LIN {X 0,Y 228.95,Z 464.335,A -85,B 0,C 180,E1 -20820.068,E2 -20820.068} C_VEL
LIN {X 0,Y 225.783,Z 455.816,A -85,B 0,C 180,E1 -20821.561,E2 -20821.561} C_VEL
LIN {X 0,Y 220.745,Z 444.883,A -85,B 0,C 180,E1 -20823.412,E2 -20823.412} C_VEL
LIN {X 0,Y 215.443,Z 435.104,A -85,B 0,C 180,E1 -20825.049,E2 -20825.049} C_VEL
LIN {X 0,Y 214.125,Z 432.902,A -85,B 0,C 180,E1 -20825.41,E2 -20825.41} C_VEL
LIN {X 0,Y 213.741,Z 431.362,A -85,B 0,C 180,E1 -20825.591,E2 -20825.591} C_VEL
LIN {X 0,Y 213.731,Z 431.362,A -85,B 0,C 180,E1 -20828.664,E2 -20828.664} C_VEL
LIN {X 0,Y 213.704,Z 431.366,A -85,B 0,C 180,E1 -20833.678,E2 -20833.678} C_VEL
LIN {X 0,Y 213.702,Z 431.365,A -85,B 0,C 180,E1 -20836.344,E2 -20836.344} C_VEL
LIN {X 0,Y 213.712,Z 431.364,A -85,B 0,C 180,E1 -20839.143,E2 -20839.143} C_VEL
LIN {X 0,Y 213.738,Z 431.359,A -85,B 0,C 180,E1 -20843.712,E2 -20843.712} C_VEL
LIN {X 0,Y 213.79,Z 431.354,A -85,B 0,C 180,E1 -20848.725,E2 -20848.725} C_VEL
LIN {X 0,Y 213.821,Z 431.351,A -85,B 0,C 180,E1 -20852.604,E2 -20852.604} C_VEL
LIN {X 0,Y 213.847,Z 431.347,A -85,B 0,C 180,E1 -20856.954,E2 -20856.954} C_VEL
LIN {X 0,Y 213.957,Z 431.335,A -85,B 0,C 180,E1 -20862.806,E2 -20862.806} C_VEL
LIN {X 0,Y 213.947,Z 431.333,A -85,B 0,C 180,E1 -20866.707,E2 -20866.707} C_VEL
LIN {X 0,Y 214.137,Z 431.305,A -85,B 0,C 180,E1 -20870.556,E2 -20870.556} C_VEL
LIN {X 0,Y 214.096,Z 431.314,A -85,B 0,C 180,E1 -20874.349,E2 -20874.349} C_VEL
LIN {X 0,Y 214.44,Z 431.245,A -85,B 0,C 180,E1 -20878.123,E2 -20878.123} C_VEL
LIN {X 0,Y 214.545,Z 431.244,A -85,B 0,C 180,E1 -20880.001,E2 -20880.001} C_VEL
LIN {X 0,Y 214.441,Z 431.269,A -85,B 0,C 180,E1 -20881.879,E2 -20881.879} C_VEL
LIN {X 0,Y 214.194,Z 431.304,A -85,B 0,C 180,E1 -20887.543,E2 -20887.543} C_VEL
LIN {X 0,Y 213.995,Z 431.329,A -85,B 0,C 180,E1 -20891.366,E2 -20891.366} C_VEL
LIN {X 0,Y 213.926,Z 431.338,A -85,B 0,C 180,E1 -20895.238,E2 -20895.238} C_VEL
LIN {X 0,Y 213.832,Z 431.349,A -85,B 0,C 180,E1 -20899.189,E2 -20899.189} C_VEL
LIN {X 0,Y 213.809,Z 431.355,A -85,B 0,C 180,E1 -20903.232,E2 -20903.232} C_VEL
LIN {X 0,Y 213.846,Z 431.557,A -85,B 0,C 180,E1 -20907.461,E2 -20907.461} C_VEL
LIN {X 0,Y 214.012,Z 433.205,A -85,B 0,C 180,E1 -20911.698,E2 -20911.698} C_VEL
LIN {X 0,Y 214.268,Z 435.135,A -85,B 0,C 180,E1 -20916.187,E2 -20916.187} C_VEL
LIN {X 0,Y 214.637,Z 437.558,A -85,B 0,C 180,E1 -20921.142,E2 -20921.142} C_VEL
LIN {X 0,Y 214.751,Z 439.049,A -85,B 0,C 180,E1 -20923.949,E2 -20923.949} C_VEL
LIN {X 0,Y 214.709,Z 440.54,A -85,B 0,C 180,E1 -20926.578,E2 -20926.578} C_VEL
LIN {X 0,Y 214.485,Z 442.03,A -85,B 0,C 180,E1 -20929.056,E2 -20929.056} C_VEL
LIN {X 0,Y 214.086,Z 443.875,A -85,B 0,C 180,E1 -20931.988,E2 -20931.988} C_VEL
LIN {X 0,Y 213.633,Z 445.658,A -85,B 0,C 180,E1 -20934.669,E2 -20934.669} C_VEL
LIN {X 0,Y 214.482,Z 448.767,A -85,B 0,C 180,E1 -20935.005,E2 -20935.005} C_VEL
LIN {X 0,Y 216.666,Z 454.962,A -85,B 0,C 180,E1 -20935.878,E2 -20935.878} C_VEL
LIN {X 0,Y 219.161,Z 463.344,A -85,B 0,C 180,E1 -20937.069,E2 -20937.069} C_VEL
LIN {X 0,Y 221.554,Z 473.865,A -85,B 0,C 180,E1 -20938.668,E2 -20938.668} C_VEL
LIN {X 0,Y 222.983,Z 483.529,A -85,B 0,C 180,E1 -20940.26,E2 -20940.26} C_VEL
LIN {X 0,Y 223.821,Z 492.472,A -85,B 0,C 180,E1 -20941.901,E2 -20941.901} C_VEL
LIN {X 0,Y 223.91,Z 501.294,A -85,B 0,C 180,E1 -20943.689,E2 -20943.689} C_VEL
LIN {X 0,Y 223.656,Z 504.689,A -85,B 0,C 180,E1 -20944.402,E2 -20944.402} C_VEL
LIN {X 0,Y 220.986,Z 514.268,A -85,B 0,C 180,E1 -20946.576,E2 -20946.576} C_VEL
LIN {X 0,Y 218.846,Z 521.593,A -85,B 0,C 180,E1 -20948.641,E2 -20948.641} C_VEL
LIN {X 0,Y 216.772,Z 528.635,A -85,B 0,C 180,E1 -20951.083,E2 -20951.083} C_VEL
LIN {X 0,Y 215.461,Z 533.139,A -85,B 0,C 180,E1 -20952.929,E2 -20952.929} C_VEL
LIN {X 0,Y 213.707,Z 538.674,A -85,B 0,C 180,E1 -20955.749,E2 -20955.749} C_VEL
LIN {X 0,Y 212.4,Z 541.079,A -85,B 0,C 180,E1 -20957.173,E2 -20957.173} C_VEL
LIN {X 0,Y 208.716,Z 544.319,A -85,B 0,C 180,E1 -20959.521,E2 -20959.521} C_VEL
LIN {X 0,Y 205.844,Z 546.363,A -85,B 0,C 180,E1 -20961.49,E2 -20961.49} C_VEL
LIN {X 0,Y 204.575,Z 547.716,A -85,B 0,C 180,E1 -20963.064,E2 -20963.064} C_VEL
LIN {X 0,Y 204.437,Z 547.992,A -85,B 0,C 180,E1 -20963.604,E2 -20963.604} C_VEL
LIN {X 0,Y 204.339,Z 549.391,A -85,B 0,C 180,E1 -20966.056,E2 -20966.056} C_VEL
LIN {X 0,Y 204.335,Z 549.984,A -85,B 0,C 180,E1 -20968.029,E2 -20968.029} C_VEL
LIN {X 0,Y 204.444,Z 550.143,A -85,B 0,C 180,E1 -20970,E2 -20970} C_VEL
LIN {X 0,Y 204.334,Z 549.984,A -85,B 0,C 180,E1 -20971.971,E2 -20971.971} C_VEL
LIN {X 0,Y 204.299,Z 549.39,A -85,B 0,C 180,E1 -20973.945,E2 -20973.945} C_VEL
LIN {X 0,Y 204.645,Z 546.935,A -85,B 0,C 180,E1 -20977.895,E2 -20977.895} C_VEL
LIN {X 0,Y 205.321,Z 543.98,A -85,B 0,C 180,E1 -20980.851,E2 -20980.851} C_VEL
LIN {X 0,Y 206.335,Z 539.986,A -85,B 0,C 180,E1 -20983.793,E2 -20983.793} C_VEL
LIN {X 0,Y 207.988,Z 534.856,A -85,B 0,C 180,E1 -20986.691,E2 -20986.691} C_VEL
LIN {X 0,Y 209.661,Z 529.593,A -85,B 0,C 180,E1 -20989.076,E2 -20989.076} C_VEL
LIN {X 0,Y 211.328,Z 524.655,A -85,B 0,C 180,E1 -20990.947,E2 -20990.947} C_VEL
LIN {X 0,Y 213.4,Z 517.322,A -85,B 0,C 180,E1 -20993.278,E2 -20993.278} C_VEL
LIN {X 0,Y 215.512,Z 510.399,A -85,B 0,C 180,E1 -20995.083,E2 -20995.083} C_VEL
LIN {X 0,Y 217.206,Z 504.49,A -85,B 0,C 180,E1 -20996.416,E2 -20996.416} C_VEL
LIN {X 0,Y 217.303,Z 494.811,A -85,B 0,C 180,E1 -20998.526,E2 -20998.526} C_VEL
LIN {X 0,Y 216.575,Z 485.637,A -85,B 0,C 180,E1 -21000.333,E2 -21000.333} C_VEL
LIN {X 0,Y 215.38,Z 476.429,A -85,B 0,C 180,E1 -21001.96,E2 -21001.96} C_VEL
LIN {X 0,Y 213.251,Z 466.398,A -85,B 0,C 180,E1 -21003.609,E2 -21003.609} C_VEL
LIN {X 0,Y 210.509,Z 456.533,A -85,B 0,C 180,E1 -21005.117,E2 -21005.117} C_VEL
LIN {X 0,Y 207.828,Z 448.996,A -85,B 0,C 180,E1 -21006.261,E2 -21006.261} C_VEL
LIN {X 0,Y 206.874,Z 446.301,A -85,B 0,C 180,E1 -21006.61,E2 -21006.61} C_VEL
LIN {X 0,Y 206.779,Z 445.482,A -85,B 0,C 180,E1 -21006.726,E2 -21006.726} C_VEL
LIN {X 0,Y 207.262,Z 443.315,A -85,B 0,C 180,E1 -21010.11,E2 -21010.11} C_VEL
LIN {X 0,Y 207.548,Z 441.811,A -85,B 0,C 180,E1 -21012.627,E2 -21012.627} C_VEL
LIN {X 0,Y 207.693,Z 440.333,A -85,B 0,C 180,E1 -21015.283,E2 -21015.283} C_VEL
LIN {X 0,Y 207.5,Z 437.944,A -85,B 0,C 180,E1 -21019.943,E2 -21019.943} C_VEL
LIN {X 0,Y 207.199,Z 435.719,A -85,B 0,C 180,E1 -21024.785,E2 -21024.785} C_VEL
LIN {X 0,Y 206.948,Z 433.839,A -85,B 0,C 180,E1 -21029.375,E2 -21029.375} C_VEL
LIN {X 0,Y 206.73,Z 432.247,A -85,B 0,C 180,E1 -21033.771,E2 -21033.771} C_VEL
LIN {X 0,Y 206.736,Z 432.236,A -85,B 0,C 180,E1 -21038.04,E2 -21038.04} C_VEL
LIN {X 0,Y 206.87,Z 432.218,A -85,B 0,C 180,E1 -21042.195,E2 -21042.195} C_VEL
LIN {X 0,Y 206.889,Z 432.214,A -85,B 0,C 180,E1 -21046.243,E2 -21046.243} C_VEL
LIN {X 0,Y 207.096,Z 432.188,A -85,B 0,C 180,E1 -21050.23,E2 -21050.23} C_VEL
LIN {X 0,Y 207.058,Z 432.192,A -85,B 0,C 180,E1 -21054.155,E2 -21054.155} C_VEL
LIN {X 0,Y 207.378,Z 432.149,A -85,B 0,C 180,E1 -21058.057,E2 -21058.057} C_VEL
LIN {X 0,Y 207.51,Z 432.119,A -85,B 0,C 180,E1 -21059.999,E2 -21059.999} C_VEL
LIN {X 0,Y 207.377,Z 432.124,A -85,B 0,C 180,E1 -21061.941,E2 -21061.941} C_VEL
LIN {X 0,Y 207.144,Z 432.18,A -85,B 0,C 180,E1 -21067.799,E2 -21067.799} C_VEL
LIN {X 0,Y 206.919,Z 432.21,A -85,B 0,C 180,E1 -21071.758,E2 -21071.758} C_VEL
LIN {X 0,Y 206.866,Z 432.214,A -85,B 0,C 180,E1 -21075.77,E2 -21075.77} C_VEL
LIN {X 0,Y 206.779,Z 432.22,A -85,B 0,C 180,E1 -21079.868,E2 -21079.868} C_VEL
LIN {X 0,Y 206.759,Z 432.226,A -85,B 0,C 180,E1 -21084.071,E2 -21084.071} C_VEL
LIN {X 0,Y 206.739,Z 432.232,A -85,B 0,C 180,E1 -21088.418,E2 -21088.418} C_VEL
LIN {X 0,Y 206.704,Z 432.237,A -85,B 0,C 180,E1 -21092.955,E2 -21092.955} C_VEL
LIN {X 0,Y 206.721,Z 432.233,A -85,B 0,C 180,E1 -21097.73,E2 -21097.73} C_VEL
LIN {X 0,Y 206.721,Z 432.235,A -85,B 0,C 180,E1 -21101.589,E2 -21101.589} C_VEL
LIN {X 0,Y 206.669,Z 432.241,A -85,B 0,C 180,E1 -21105.57,E2 -21105.57} C_VEL
LIN {X 0,Y 206.669,Z 432.24,A -85,B 0,C 180,E1 -21109.752,E2 -21109.752} C_VEL
LIN {X 0,Y 206.71,Z 432.237,A -85,B 0,C 180,E1 -21113.049,E2 -21113.049} C_VEL
LIN {X 0,Y 207.757,Z 435.179,A -85,B 0,C 180,E1 -21113.464,E2 -21113.464} C_VEL
LIN {X 0,Y 209.142,Z 437.168,A -85,B 0,C 180,E1 -21113.858,E2 -21113.858} C_VEL
LIN {X 0,Y 214.876,Z 447.881,A -85,B 0,C 180,E1 -21115.778,E2 -21115.778} C_VEL
LIN {X 0,Y 220.603,Z 460.836,A -85,B 0,C 180,E1 -21118.167,E2 -21118.167} C_VEL
LIN {X 0,Y 223.937,Z 470.772,A -85,B 0,C 180,E1 -21120.071,E2 -21120.071} C_VEL
LIN {X 0,Y 226.919,Z 479.248,A -85,B 0,C 180,E1 -21121.902,E2 -21121.902} C_VEL
LIN {X 0,Y 230.977,Z 487.85,A -85,B 0,C 180,E1 -21124.091,E2 -21124.091} C_VEL
LIN {X 0,Y 235.85,Z 495.643,A -85,B 0,C 180,E1 -21126.388,E2 -21126.388} C_VEL
LIN {X 0,Y 242.584,Z 503.921,A -85,B 0,C 180,E1 -21129.183,E2 -21129.183} C_VEL
LIN {X 0,Y 250.878,Z 511.914,A -85,B 0,C 180,E1 -21132.259,E2 -21132.259} C_VEL
LIN {X 0,Y 258.464,Z 517.884,A -85,B 0,C 180,E1 -21134.854,E2 -21134.854} C_VEL
LIN {X 0,Y 267.452,Z 523.982,A -85,B 0,C 180,E1 -21137.865,E2 -21137.865} C_VEL
LIN {X 0,Y 274.679,Z 528.41,A -85,B 0,C 180,E1 -21140.427,E2 -21140.427} C_VEL
LIN {X 0,Y 280.649,Z 531.794,A -85,B 0,C 180,E1 -21142.807,E2 -21142.807} C_VEL
LIN {X 0,Y 283.647,Z 533.508,A -85,B 0,C 180,E1 -21144.312,E2 -21144.312} C_VEL
LIN {X 0,Y 285.796,Z 534.827,A -85,B 0,C 180,E1 -21145.769,E2 -21145.769} C_VEL
LIN {X 0,Y 288.397,Z 535.966,A -85,B 0,C 180,E1 -21147.597,E2 -21147.597} C_VEL
LIN {X 0,Y 289.489,Z 536.314,A -85,B 0,C 180,E1 -21148.609,E2 -21148.609} C_VEL
LIN {X 0,Y 290.513,Z 536.484,A -85,B 0,C 180,E1 -21150,E2 -21150} C_VEL
LIN {X 0,Y 289.482,Z 536.314,A -85,B 0,C 180,E1 -21151.391,E2 -21151.391} C_VEL
LIN {X 0,Y 287.845,Z 535.767,A -85,B 0,C 180,E1 -21152.799,E2 -21152.799} C_VEL
LIN {X 0,Y 285.796,Z 534.827,A -85,B 0,C 180,E1 -21154.231,E2 -21154.231} C_VEL
LIN {X 0,Y 282.767,Z 532.973,A -85,B 0,C 180,E1 -21156.196,E2 -21156.196} C_VEL
LIN {X 0,Y 280.611,Z 531.795,A -85,B 0,C 180,E1 -21157.194,E2 -21157.194} C_VEL
LIN {X 0,Y 274.692,Z 528.41,A -85,B 0,C 180,E1 -21159.573,E2 -21159.573} C_VEL
LIN {X 0,Y 267.467,Z 523.982,A -85,B 0,C 180,E1 -21162.134,E2 -21162.134} C_VEL
LIN {X 0,Y 258.459,Z 517.897,A -85,B 0,C 180,E1 -21165.142,E2 -21165.142} C_VEL
LIN {X 0,Y 250.189,Z 511.27,A -85,B 0,C 180,E1 -21167.998,E2 -21167.998} C_VEL
LIN {X 0,Y 242.6,Z 503.901,A -85,B 0,C 180,E1 -21170.821,E2 -21170.821} C_VEL
LIN {X 0,Y 235.851,Z 495.641,A -85,B 0,C 180,E1 -21173.612,E2 -21173.612} C_VEL
LIN {X 0,Y 230.442,Z 486.799,A -85,B 0,C 180,E1 -21176.187,E2 -21176.187} C_VEL
LIN {X 0,Y 226.499,Z 478.07,A -85,B 0,C 180,E1 -21178.368,E2 -21178.368} C_VEL
LIN {X 0,Y 222.715,Z 466.813,A -85,B 0,C 180,E1 -21180.697,E2 -21180.697} C_VEL
LIN {X 0,Y 219.268,Z 457.558,A -85,B 0,C 180,E1 -21182.446,E2 -21182.446} C_VEL
LIN {X 0,Y 214.039,Z 446.14,A -85,B 0,C 180,E1 -21184.519,E2 -21184.519} C_VEL
LIN {X 0,Y 208.408,Z 436.025,A -85,B 0,C 180,E1 -21186.376,E2 -21186.376} C_VEL
LIN {X 0,Y 206.986,Z 433.495,A -85,B 0,C 180,E1 -21186.81,E2 -21186.81} C_VEL
LIN {X 0,Y 206.695,Z 432.239,A -85,B 0,C 180,E1 -21186.946,E2 -21186.946} C_VEL
LIN {X 0,Y 206.641,Z 432.246,A -85,B 0,C 180,E1 -21191.564,E2 -21191.564} C_VEL
LIN {X 0,Y 206.63,Z 432.247,A -85,B 0,C 180,E1 -21195.582,E2 -21195.582} C_VEL
LIN {X 0,Y 206.655,Z 432.243,A -85,B 0,C 180,E1 -21199.749,E2 -21199.749} C_VEL
LIN {X 0,Y 206.694,Z 432.237,A -85,B 0,C 180,E1 -21204.689,E2 -21204.689} C_VEL
LIN {X 0,Y 206.718,Z 432.236,A -85,B 0,C 180,E1 -21209.34,E2 -21209.34} C_VEL
LIN {X 0,Y 206.728,Z 432.231,A -85,B 0,C 180,E1 -21213.773,E2 -21213.773} C_VEL
LIN {X 0,Y 206.753,Z 432.23,A -85,B 0,C 180,E1 -21218.044,E2 -21218.044} C_VEL
LIN {X 0,Y 206.868,Z 432.215,A -85,B 0,C 180,E1 -21222.197,E2 -21222.197} C_VEL
LIN {X 0,Y 206.889,Z 432.209,A -85,B 0,C 180,E1 -21226.245,E2 -21226.245} C_VEL
LIN {X 0,Y 207.095,Z 432.182,A -85,B 0,C 180,E1 -21230.232,E2 -21230.232} C_VEL
LIN {X 0,Y 207.057,Z 432.193,A -85,B 0,C 180,E1 -21234.157,E2 -21234.157} C_VEL
LIN {X 0,Y 207.377,Z 432.124,A -85,B 0,C 180,E1 -21238.059,E2 -21238.059} C_VEL
LIN {X 0,Y 207.51,Z 432.119,A -85,B 0,C 180,E1 -21240.001,E2 -21240.001} C_VEL
LIN {X 0,Y 207.378,Z 432.149,A -85,B 0,C 180,E1 -21241.943,E2 -21241.943} C_VEL
LIN {X 0,Y 207.137,Z 432.183,A -85,B 0,C 180,E1 -21247.801,E2 -21247.801} C_VEL
LIN {X 0,Y 206.92,Z 432.211,A -85,B 0,C 180,E1 -21251.76,E2 -21251.76} C_VEL
LIN {X 0,Y 206.861,Z 432.22,A -85,B 0,C 180,E1 -21255.772,E2 -21255.772} C_VEL
LIN {X 0,Y 206.775,Z 432.229,A -85,B 0,C 180,E1 -21259.871,E2 -21259.871} C_VEL
LIN {X 0,Y 206.745,Z 432.238,A -85,B 0,C 180,E1 -21264.076,E2 -21264.076} C_VEL
LIN {X 0,Y 206.73,Z 432.253,A -85,B 0,C 180,E1 -21266.229,E2 -21266.229} C_VEL
LIN {X 0,Y 206.948,Z 433.841,A -85,B 0,C 180,E1 -21270.625,E2 -21270.625} C_VEL
LIN {X 0,Y 207.206,Z 435.844,A -85,B 0,C 180,E1 -21275.51,E2 -21275.51} C_VEL
LIN {X 0,Y 207.505,Z 437.945,A -85,B 0,C 180,E1 -21280.055,E2 -21280.055} C_VEL
LIN {X 0,Y 207.632,Z 439.227,A -85,B 0,C 180,E1 -21282.608,E2 -21282.608} C_VEL
LIN {X 0,Y 207.678,Z 440.668,A -85,B 0,C 180,E1 -21285.29,E2 -21285.29} C_VEL
LIN {X 0,Y 207.479,Z 442.319,A -85,B 0,C 180,E1 -21288.179,E2 -21288.179} C_VEL
LIN {X 0,Y 206.932,Z 444.794,A -85,B 0,C 180,E1 -21292.315,E2 -21292.315} C_VEL
LIN {X 0,Y 206.779,Z 445.439,A -85,B 0,C 180,E1 -21293.275,E2 -21293.275} C_VEL
LIN {X 0,Y 207.828,Z 448.982,A -85,B 0,C 180,E1 -21293.738,E2 -21293.738} C_VEL
LIN {X 0,Y 211.592,Z 459.902,A -85,B 0,C 180,E1 -21295.378,E2 -21295.378} C_VEL
LIN {X 0,Y 214.365,Z 471.313,A -85,B 0,C 180,E1 -21297.172,E2 -21297.172} C_VEL
LIN {X 0,Y 216.106,Z 481.185,A -85,B 0,C 180,E1 -21298.862,E2 -21298.862} C_VEL
LIN {X 0,Y 217.044,Z 490.271,A -85,B 0,C 180,E1 -21300.554,E2 -21300.554} C_VEL
LIN {X 0,Y 217.32,Z 498.233,A -85,B 0,C 180,E1 -21302.174,E2 -21302.174} C_VEL
LIN {X 0,Y 216.968,Z 505.58,A -85,B 0,C 180,E1 -21303.811,E2 -21303.811} C_VEL
LIN {X 0,Y 214.482,Z 514.07,A -85,B 0,C 180,E1 -21305.821,E2 -21305.821} C_VEL
LIN {X 0,Y 212.042,Z 521.97,A -85,B 0,C 180,E1 -21308.134,E2 -21308.134} C_VEL
LIN {X 0,Y 210.053,Z 528.438,A -85,B 0,C 180,E1 -21310.453,E2 -21310.453} C_VEL
LIN {X 0,Y 208.659,Z 532.941,A -85,B 0,C 180,E1 -21312.354,E2 -21312.354} C_VEL
LIN {X 0,Y 206.707,Z 538.795,A -85,B 0,C 180,E1 -21315.462,E2 -21315.462} C_VEL
LIN {X 0,Y 205.611,Z 542.761,A -85,B 0,C 180,E1 -21318.166,E2 -21318.166} C_VEL
LIN {X 0,Y 205.071,Z 545.133,A -85,B 0,C 180,E1 -21320.134,E2 -21320.134} C_VEL
LIN {X 0,Y 204.437,Z 547.992,A -85,B 0,C 180,E1 -21323.604,E2 -21323.604} C_VEL
LIN {X 0,Y 203.673,Z 549.008,A -85,B 0,C 180,E1 -21325.226,E2 -21325.226} C_VEL
LIN {X 0,Y 202.069,Z 549.675,A -85,B 0,C 180,E1 -21326.833,E2 -21326.833} C_VEL
LIN {X 0,Y 198.386,Z 550.084,A -85,B 0,C 180,E1 -21330.102,E2 -21330.102} C_VEL
LIN {X 0,Y 197.324,Z 549.856,A -85,B 0,C 180,E1 -21331.809,E2 -21331.809} C_VEL
LIN {X 0,Y 197.219,Z 549.687,A -85,B 0,C 180,E1 -21332.386,E2 -21332.386} C_VEL
LIN {X 0,Y 197.21,Z 549.193,A -85,B 0,C 180,E1 -21334.087,E2 -21334.087} C_VEL
LIN {X 0,Y 197.595,Z 546.737,A -85,B 0,C 180,E1 -21338.179,E2 -21338.179} C_VEL
LIN {X 0,Y 198.307,Z 543.782,A -85,B 0,C 180,E1 -21341.24,E2 -21341.24} C_VEL
LIN {X 0,Y 199.408,Z 539.788,A -85,B 0,C 180,E1 -21344.283,E2 -21344.283} C_VEL
LIN {X 0,Y 201.169,Z 534.658,A -85,B 0,C 180,E1 -21347.274,E2 -21347.274} C_VEL
LIN {X 0,Y 202.94,Z 529.395,A -85,B 0,C 180,E1 -21349.733,E2 -21349.733} C_VEL
LIN {X 0,Y 204.659,Z 524.456,A -85,B 0,C 180,E1 -21351.663,E2 -21351.663} C_VEL
LIN {X 0,Y 206.363,Z 518.752,A -85,B 0,C 180,E1 -21353.587,E2 -21353.587} C_VEL
LIN {X 0,Y 209.076,Z 510.201,A -85,B 0,C 180,E1 -21355.911,E2 -21355.911} C_VEL
LIN {X 0,Y 210.544,Z 505.38,A -85,B 0,C 180,E1 -21357.052,E2 -21357.052} C_VEL
LIN {X 0,Y 210.696,Z 494.601,A -85,B 0,C 180,E1 -21359.508,E2 -21359.508} C_VEL
LIN {X 0,Y 209.952,Z 484.831,A -85,B 0,C 180,E1 -21361.498,E2 -21361.498} C_VEL
LIN {X 0,Y 208.694,Z 476.106,A -85,B 0,C 180,E1 -21363.128,E2 -21363.128} C_VEL
LIN {X 0,Y 206.665,Z 466.416,A -85,B 0,C 180,E1 -21364.804,E2 -21364.804} C_VEL
LIN {X 0,Y 203.784,Z 456.5,A -85,B 0,C 180,E1 -21366.44,E2 -21366.44} C_VEL
LIN {X 0,Y 201.057,Z 448.967,A -85,B 0,C 180,E1 -21367.675,E2 -21367.675} C_VEL
LIN {X 0,Y 200.078,Z 446.209,A -85,B 0,C 180,E1 -21368.061,E2 -21368.061} C_VEL
LIN {X 0,Y 199.968,Z 445.246,A -85,B 0,C 180,E1 -21368.243,E2 -21368.243} C_VEL
LIN {X 0,Y 200.497,Z 442.642,A -85,B 0,C 180,E1 -21372.597,E2 -21372.597} C_VEL
LIN {X 0,Y 200.63,Z 441.069,A -85,B 0,C 180,E1 -21375.524,E2 -21375.524} C_VEL
LIN {X 0,Y 200.566,Z 439.695,A -85,B 0,C 180,E1 -21378.257,E2 -21378.257} C_VEL
LIN {X 0,Y 200.388,Z 438.48,A -85,B 0,C 180,E1 -21380.853,E2 -21380.853} C_VEL
LIN {X 0,Y 200.082,Z 436.327,A -85,B 0,C 180,E1 -21385.804,E2 -21385.804} C_VEL
LIN {X 0,Y 199.872,Z 434.479,A -85,B 0,C 180,E1 -21390.509,E2 -21390.509} C_VEL
LIN {X 0,Y 199.663,Z 433.116,A -85,B 0,C 180,E1 -21395.013,E2 -21395.013} C_VEL
LIN {X 0,Y 199.688,Z 433.113,A -85,B 0,C 180,E1 -21399.392,E2 -21399.392} C_VEL
LIN {X 0,Y 199.799,Z 433.099,A -85,B 0,C 180,E1 -21403.655,E2 -21403.655} C_VEL
LIN {X 0,Y 199.87,Z 433.09,A -85,B 0,C 180,E1 -21407.819,E2 -21407.819} C_VEL
LIN {X 0,Y 200.085,Z 433.061,A -85,B 0,C 180,E1 -21411.922,E2 -21411.922} C_VEL
LIN {X 0,Y 200.317,Z 433.028,A -85,B 0,C 180,E1 -21417.988,E2 -21417.988} C_VEL
LIN {X 0,Y 200.475,Z 432.994,A -85,B 0,C 180,E1 -21419.999,E2 -21419.999} C_VEL
LIN {X 0,Y 200.023,Z 433.053,A -85,B 0,C 180,E1 -21424.028,E2 -21424.028} C_VEL
LIN {X 0,Y 200.091,Z 433.058,A -85,B 0,C 180,E1 -21428.075,E2 -21428.075} C_VEL
LIN {X 0,Y 199.869,Z 433.088,A -85,B 0,C 180,E1 -21432.178,E2 -21432.178} C_VEL
LIN {X 0,Y 199.802,Z 433.095,A -85,B 0,C 180,E1 -21436.342,E2 -21436.342} C_VEL
LIN {X 0,Y 199.695,Z 433.104,A -85,B 0,C 180,E1 -21440.605,E2 -21440.605} C_VEL
LIN {X 0,Y 199.668,Z 433.107,A -85,B 0,C 180,E1 -21444.984,E2 -21444.984} C_VEL
LIN {X 0,Y 199.67,Z 433.114,A -85,B 0,C 180,E1 -21449.522,E2 -21449.522} C_VEL
LIN {X 0,Y 199.659,Z 433.115,A -85,B 0,C 180,E1 -21452.352,E2 -21452.352} C_VEL
LIN {X 0,Y 199.649,Z 433.117,A -85,B 0,C 180,E1 -21456.756,E2 -21456.756} C_VEL
LIN {X 0,Y 199.695,Z 433.111,A -85,B 0,C 180,E1 -21459.306,E2 -21459.306} C_VEL
LIN {X 0,Y 199.659,Z 433.115,A -85,B 0,C 180,E1 -21462.338,E2 -21462.338} C_VEL
LIN {X 0,Y 199.626,Z 433.118,A -85,B 0,C 180,E1 -21465.243,E2 -21465.243} C_VEL
LIN {X 0,Y 199.637,Z 433.118,A -85,B 0,C 180,E1 -21470.756,E2 -21470.756} C_VEL
LIN {X 0,Y 199.672,Z 433.114,A -85,B 0,C 180,E1 -21471.549,E2 -21471.549} C_VEL
LIN {X 0,Y 200.765,Z 436.111,A -85,B 0,C 180,E1 -21472.012,E2 -21472.012} C_VEL
LIN {X 0,Y 202.338,Z 438.455,A -85,B 0,C 180,E1 -21472.497,E2 -21472.497} C_VEL
LIN {X 0,Y 208.631,Z 449.967,A -85,B 0,C 180,E1 -21474.779,E2 -21474.779} C_VEL
LIN {X 0,Y 213.417,Z 460.812,A -85,B 0,C 180,E1 -21476.927,E2 -21476.927} C_VEL
LIN {X 0,Y 217.071,Z 471.364,A -85,B 0,C 180,E1 -21479.086,E2 -21479.086} C_VEL
LIN {X 0,Y 219.94,Z 480.544,A -85,B 0,C 180,E1 -21481.136,E2 -21481.136} C_VEL
LIN {X 0,Y 223.953,Z 489.751,A -85,B 0,C 180,E1 -21483.592,E2 -21483.592} C_VEL
LIN {X 0,Y 228.955,Z 498.056,A -85,B 0,C 180,E1 -21486.188,E2 -21486.188} C_VEL
LIN {X 0,Y 234.114,Z 504.632,A -85,B 0,C 180,E1 -21488.527,E2 -21488.527} C_VEL
LIN {X 0,Y 241.5,Z 512.13,A -85,B 0,C 180,E1 -21491.529,E2 -21491.529} C_VEL
LIN {X 0,Y 250.543,Z 519.184,A -85,B 0,C 180,E1 -21494.77,E2 -21494.77} C_VEL
LIN {X 0,Y 258.96,Z 524.71,A -85,B 0,C 180,E1 -21497.687,E2 -21497.687} C_VEL
LIN {X 0,Y 266.352,Z 528.907,A -85,B 0,C 180,E1 -21500.276,E2 -21500.276} C_VEL
LIN {X 0,Y 272.29,Z 532.028,A -85,B 0,C 180,E1 -21502.585,E2 -21502.585} C_VEL
LIN {X 0,Y 275.869,Z 533.726,A -85,B 0,C 180,E1 -21504.151,E2 -21504.151} C_VEL
LIN {X 0,Y 278.242,Z 535.036,A -85,B 0,C 180,E1 -21505.654,E2 -21505.654} C_VEL
LIN {X 0,Y 281.323,Z 536.263,A -85,B 0,C 180,E1 -21507.798,E2 -21507.798} C_VEL
LIN {X 0,Y 282.198,Z 536.515,A -85,B 0,C 180,E1 -21508.573,E2 -21508.573} C_VEL
LIN {X 0,Y 283.347,Z 536.679,A -85,B 0,C 180,E1 -21510,E2 -21510} C_VEL
LIN {X 0,Y 282.194,Z 536.515,A -85,B 0,C 180,E1 -21511.427,E2 -21511.427} C_VEL
LIN {X 0,Y 280.345,Z 535.976,A -85,B 0,C 180,E1 -21512.874,E2 -21512.874} C_VEL
LIN {X 0,Y 278.24,Z 535.036,A -85,B 0,C 180,E1 -21514.346,E2 -21514.346} C_VEL
LIN {X 0,Y 275.579,Z 533.618,A -85,B 0,C 180,E1 -21515.964,E2 -21515.964} C_VEL
LIN {X 0,Y 269.934,Z 530.805,A -85,B 0,C 180,E1 -21518.369,E2 -21518.369} C_VEL
LIN {X 0,Y 264.389,Z 527.859,A -85,B 0,C 180,E1 -21520.417,E2 -21520.417} C_VEL
LIN {X 0,Y 258.186,Z 524.247,A -85,B 0,C 180,E1 -21522.578,E2 -21522.578} C_VEL
LIN {X 0,Y 250.516,Z 519.224,A -85,B 0,C 180,E1 -21525.216,E2 -21525.216} C_VEL
LIN {X 0,Y 242.22,Z 512.669,A -85,B 0,C 180,E1 -21528.233,E2 -21528.233} C_VEL
LIN {X 0,Y 235.17,Z 505.849,A -85,B 0,C 180,E1 -21531.015,E2 -21531.015} C_VEL
LIN {X 0,Y 229.748,Z 499.19,A -85,B 0,C 180,E1 -21533.432,E2 -21533.432} C_VEL
LIN {X 0,Y 224.826,Z 491.276,A -85,B 0,C 180,E1 -21535.952,E2 -21535.952} C_VEL
LIN {X 0,Y 221.187,Z 483.619,A -85,B 0,C 180,E1 -21538.083,E2 -21538.083} C_VEL
LIN {X 0,Y 218.121,Z 474.859,A -85,B 0,C 180,E1 -21540.164,E2 -21540.164} C_VEL
LIN {X 0,Y 215.006,Z 465.027,A -85,B 0,C 180,E1 -21542.207,E2 -21542.207} C_VEL
LIN {X 0,Y 211.104,Z 455.426,A -85,B 0,C 180,E1 -21544.137,E2 -21544.137} C_VEL
LIN {X 0,Y 206.803,Z 446.534,A -85,B 0,C 180,E1 -21545.895,E2 -21545.895} C_VEL
LIN {X 0,Y 202.025,Z 437.714,A -85,B 0,C 180,E1 -21547.627,E2 -21547.627} C_VEL
LIN {X 0,Y 200.071,Z 434.776,A -85,B 0,C 180,E1 -21548.25,E2 -21548.25} C_VEL
LIN {X 0,Y 199.676,Z 433.113,A -85,B 0,C 180,E1 -21548.505,E2 -21548.505} C_VEL
LIN {X 0,Y 199.573,Z 433.125,A -85,B 0,C 180,E1 -21552.311,E2 -21552.311} C_VEL
LIN {X 0,Y 199.576,Z 433.124,A -85,B 0,C 180,E1 -21555.229,E2 -21555.229} C_VEL
LIN {X 0,Y 199.575,Z 433.125,A -85,B 0,C 180,E1 -21558.005,E2 -21558.005} C_VEL
LIN {X 0,Y 199.605,Z 433.122,A -85,B 0,C 180,E1 -21560.768,E2 -21560.768} C_VEL
LIN {X 0,Y 199.608,Z 433.12,A -85,B 0,C 180,E1 -21565.714,E2 -21565.714} C_VEL
LIN {X 0,Y 199.696,Z 433.11,A -85,B 0,C 180,E1 -21568.138,E2 -21568.138} C_VEL
LIN {X 0,Y 199.682,Z 433.113,A -85,B 0,C 180,E1 -21572.772,E2 -21572.772} C_VEL
LIN {X 0,Y 199.733,Z 433.106,A -85,B 0,C 180,E1 -21577.23,E2 -21577.23} C_VEL
LIN {X 0,Y 199.792,Z 433.096,A -85,B 0,C 180,E1 -21581.759,E2 -21581.759} C_VEL
LIN {X 0,Y 199.831,Z 433.087,A -85,B 0,C 180,E1 -21585.749,E2 -21585.749} C_VEL
LIN {X 0,Y 200.018,Z 433.064,A -85,B 0,C 180,E1 -21589.883,E2 -21589.883} C_VEL
LIN {X 0,Y 200.018,Z 433.069,A -85,B 0,C 180,E1 -21593.95,E2 -21593.95} C_VEL
LIN {X 0,Y 200.316,Z 433.002,A -85,B 0,C 180,E1 -21597.991,E2 -21597.991} C_VEL
LIN {X 0,Y 200.475,Z 432.994,A -85,B 0,C 180,E1 -21600.001,E2 -21600.001} C_VEL
LIN {X 0,Y 200.024,Z 433.07,A -85,B 0,C 180,E1 -21604.031,E2 -21604.031} C_VEL
LIN {X 0,Y 200.085,Z 433.063,A -85,B 0,C 180,E1 -21608.078,E2 -21608.078} C_VEL
LIN {X 0,Y 199.87,Z 433.092,A -85,B 0,C 180,E1 -21612.181,E2 -21612.181} C_VEL
LIN {X 0,Y 199.799,Z 433.099,A -85,B 0,C 180,E1 -21616.345,E2 -21616.345} C_VEL
LIN {X 0,Y 199.688,Z 433.112,A -85,B 0,C 180,E1 -21620.608,E2 -21620.608} C_VEL
LIN {X 0,Y 199.663,Z 433.117,A -85,B 0,C 180,E1 -21624.987,E2 -21624.987} C_VEL
LIN {X 0,Y 199.872,Z 434.478,A -85,B 0,C 180,E1 -21629.491,E2 -21629.491} C_VEL
LIN {X 0,Y 200.082,Z 436.316,A -85,B 0,C 180,E1 -21634.196,E2 -21634.196} C_VEL
LIN {X 0,Y 200.424,Z 438.645,A -85,B 0,C 180,E1 -21639.518,E2 -21639.518} C_VEL
LIN {X 0,Y 200.587,Z 440.143,A -85,B 0,C 180,E1 -21642.628,E2 -21642.628} C_VEL
LIN {X 0,Y 200.611,Z 441.649,A -85,B 0,C 180,E1 -21645.521,E2 -21645.521} C_VEL
LIN {X 0,Y 200.401,Z 443.132,A -85,B 0,C 180,E1 -21648.217,E2 -21648.217} C_VEL
LIN {X 0,Y 199.959,Z 445.248,A -85,B 0,C 180,E1 -21651.813,E2 -21651.813} C_VEL
LIN {X 0,Y 200.938,Z 448.686,A -85,B 0,C 180,E1 -21652.279,E2 -21652.279} C_VEL
LIN {X 0,Y 202.011,Z 451.529,A -85,B 0,C 180,E1 -21652.751,E2 -21652.751} C_VEL
LIN {X 0,Y 205.019,Z 460.093,A -85,B 0,C 180,E1 -21654.147,E2 -21654.147} C_VEL
LIN {X 0,Y 207.566,Z 470.252,A -85,B 0,C 180,E1 -21655.832,E2 -21655.832} C_VEL
LIN {X 0,Y 209.479,Z 480.91,A -85,B 0,C 180,E1 -21657.75,E2 -21657.75} C_VEL
LIN {X 0,Y 210.472,Z 490.944,A -85,B 0,C 180,E1 -21659.719,E2 -21659.719} C_VEL
LIN {X 0,Y 210.748,Z 498.523,A -85,B 0,C 180,E1 -21661.345,E2 -21661.345} C_VEL
LIN {X 0,Y 210.298,Z 506.364,A -85,B 0,C 180,E1 -21663.183,E2 -21663.183} C_VEL
LIN {X 0,Y 207.458,Z 515.499,A -85,B 0,C 180,E1 -21665.482,E2 -21665.482} C_VEL
LIN {X 0,Y 205.201,Z 522.458,A -85,B 0,C 180,E1 -21667.63,E2 -21667.63} C_VEL
LIN {X 0,Y 203.368,Z 528.24,A -85,B 0,C 180,E1 -21669.783,E2 -21669.783} C_VEL
LIN {X 0,Y 201.868,Z 532.743,A -85,B 0,C 180,E1 -21671.74,E2 -21671.74} C_VEL
LIN {X 0,Y 199.93,Z 538.233,A -85,B 0,C 180,E1 -21674.714,E2 -21674.714} C_VEL
LIN {X 0,Y 198.631,Z 542.563,A -85,B 0,C 180,E1 -21677.744,E2 -21677.744} C_VEL
LIN {X 0,Y 198.042,Z 544.935,A -85,B 0,C 180,E1 -21679.78,E2 -21679.78} C_VEL
LIN {X 0,Y 197.363,Z 547.922,A -85,B 0,C 180,E1 -21683.562,E2 -21683.562} C_VEL
LIN {X 0,Y 197.244,Z 549.248,A -85,B 0,C 180,E1 -21686.102,E2 -21686.102} C_VEL
LIN {X 0,Y 197.243,Z 549.787,A -85,B 0,C 180,E1 -21687.958,E2 -21687.958} C_VEL
LIN {X 0,Y 197.345,Z 549.946,A -85,B 0,C 180,E1 -21690,E2 -21690} C_VEL
LIN {X 0,Y 197.219,Z 549.687,A -85,B 0,C 180,E1 -21692.386,E2 -21692.386} C_VEL
LIN {X 0,Y 196.526,Z 549.189,A -85,B 0,C 180,E1 -21694.086,E2 -21694.086} C_VEL
LIN {X 0,Y 193.856,Z 547.681,A -85,B 0,C 180,E1 -21696.86,E2 -21696.86} C_VEL
LIN {X 0,Y 191.8,Z 546.059,A -85,B 0,C 180,E1 -21699.101,E2 -21699.101} C_VEL
LIN {X 0,Y 191.174,Z 544.238,A -85,B 0,C 180,E1 -21701.089,E2 -21701.089} C_VEL
LIN {X 0,Y 191.231,Z 543.896,A -85,B 0,C 180,E1 -21701.371,E2 -21701.371} C_VEL
LIN {X 0,Y 192.063,Z 541.122,A -85,B 0,C 180,E1 -21703.759,E2 -21703.759} C_VEL
LIN {X 0,Y 193.69,Z 536.375,A -85,B 0,C 180,E1 -21706.874,E2 -21706.874} C_VEL
LIN {X 0,Y 195.83,Z 530.353,A -85,B 0,C 180,E1 -21709.934,E2 -21709.934} C_VEL
LIN {X 0,Y 198.06,Z 524.126,A -85,B 0,C 180,E1 -21712.476,E2 -21712.476} C_VEL
LIN {X 0,Y 199.844,Z 518.553,A -85,B 0,C 180,E1 -21714.406,E2 -21714.406} C_VEL
LIN {X 0,Y 202.706,Z 510.003,A -85,B 0,C 180,E1 -21716.789,E2 -21716.789} C_VEL
LIN {X 0,Y 203.864,Z 506.164,A -85,B 0,C 180,E1 -21717.735,E2 -21717.735} C_VEL
LIN {X 0,Y 204.181,Z 495.705,A -85,B 0,C 180,E1 -21720.272,E2 -21720.272} C_VEL
LIN {X 0,Y 203.513,Z 485.672,A -85,B 0,C 180,E1 -21722.428,E2 -21722.428} C_VEL
LIN {X 0,Y 202.213,Z 476.563,A -85,B 0,C 180,E1 -21724.234,E2 -21724.234} C_VEL
LIN {X 0,Y 200.089,Z 466.295,A -85,B 0,C 180,E1 -21726.111,E2 -21726.111} C_VEL
LIN {X 0,Y 196.974,Z 456.129,A -85,B 0,C 180,E1 -21727.929,E2 -21727.929} C_VEL
LIN {X 0,Y 194.257,Z 448.777,A -85,B 0,C 180,E1 -21729.236,E2 -21729.236} C_VEL
LIN {X 0,Y 193.15,Z 445.604,A -85,B 0,C 180,E1 -21729.712,E2 -21729.712} C_VEL
LIN {X 0,Y 193.089,Z 445.051,A -85,B 0,C 180,E1 -21729.817,E2 -21729.817} C_VEL
LIN {X 0,Y 193.487,Z 442.895,A -85,B 0,C 180,E1 -21733.639,E2 -21733.639} C_VEL
LIN {X 0,Y 193.544,Z 441.419,A -85,B 0,C 180,E1 -21736.571,E2 -21736.571} C_VEL
LIN {X 0,Y 193.424,Z 439.921,A -85,B 0,C 180,E1 -21739.73,E2 -21739.73} C_VEL
LIN {X 0,Y 193.122,Z 437.928,A -85,B 0,C 180,E1 -21744.389,E2 -21744.389} C_VEL
LIN {X 0,Y 192.876,Z 436.02,A -85,B 0,C 180,E1 -21749.326,E2 -21749.326} C_VEL
LIN {X 0,Y 192.826,Z 435.158,A -85,B 0,C 180,E1 -21751.717,E2 -21751.717} C_VEL
LIN {X 0,Y 192.683,Z 433.986,A -85,B 0,C 180,E1 -21756.344,E2 -21756.344} C_VEL
LIN {X 0,Y 192.729,Z 433.98,A -85,B 0,C 180,E1 -21761.457,E2 -21761.457} C_VEL
LIN {X 0,Y 192.759,Z 433.975,A -85,B 0,C 180,E1 -21765.212,E2 -21765.212} C_VEL
LIN {X 0,Y 192.942,Z 433.953,A -85,B 0,C 180,E1 -21769.565,E2 -21769.565} C_VEL
LIN {X 0,Y 192.982,Z 433.948,A -85,B 0,C 180,E1 -21773.727,E2 -21773.727} C_VEL
LIN {X 0,Y 193.259,Z 433.908,A -85,B 0,C 180,E1 -21777.915,E2 -21777.915} C_VEL
LIN {X 0,Y 193.439,Z 433.869,A -85,B 0,C 180,E1 -21779.999,E2 -21779.999} C_VEL
LIN {X 0,Y 192.969,Z 433.932,A -85,B 0,C 180,E1 -21784.176,E2 -21784.176} C_VEL
LIN {X 0,Y 193.037,Z 433.937,A -85,B 0,C 180,E1 -21788.373,E2 -21788.373} C_VEL
LIN {X 0,Y 192.797,Z 433.969,A -85,B 0,C 180,E1 -21792.632,E2 -21792.632} C_VEL
LIN {X 0,Y 192.754,Z 433.975,A -85,B 0,C 180,E1 -21796.958,E2 -21796.958} C_VEL
LIN {X 0,Y 192.632,Z 433.988,A -85,B 0,C 180,E1 -21801.396,E2 -21801.396} C_VEL
LIN {X 0,Y 192.659,Z 433.981,A -85,B 0,C 180,E1 -21804.224,E2 -21804.224} C_VEL
LIN {X 0,Y 192.645,Z 433.988,A -85,B 0,C 180,E1 -21808.891,E2 -21808.891} C_VEL
LIN {X 0,Y 192.596,Z 433.994,A -85,B 0,C 180,E1 -21813.185,E2 -21813.185} C_VEL
LIN {X 0,Y 192.608,Z 433.992,A -85,B 0,C 180,E1 -21818.337,E2 -21818.337} C_VEL
LIN {X 0,Y 192.596,Z 433.994,A -85,B 0,C 180,E1 -21823.13,E2 -21823.13} C_VEL
LIN {X 0,Y 192.535,Z 434.001,A -85,B 0,C 180,E1 -21826.889,E2 -21826.889} C_VEL
LIN {X 0,Y 192.554,Z 433.999,A -85,B 0,C 180,E1 -21829.873,E2 -21829.873} C_VEL
LIN {X 0,Y 193.641,Z 436.921,A -85,B 0,C 180,E1 -21830.382,E2 -21830.382} C_VEL
LIN {X 0,Y 195.283,Z 439.141,A -85,B 0,C 180,E1 -21830.92,E2 -21830.92} C_VEL
LIN {X 0,Y 201.468,Z 450.437,A -85,B 0,C 180,E1 -21833.351,E2 -21833.351} C_VEL
LIN {X 0,Y 206.285,Z 460.989,A -85,B 0,C 180,E1 -21835.619,E2 -21835.619} C_VEL
LIN {X 0,Y 210.105,Z 471.501,A -85,B 0,C 180,E1 -21837.928,E2 -21837.928} C_VEL
LIN {X 0,Y 213.119,Z 481.9,A -85,B 0,C 180,E1 -21840.354,E2 -21840.354} C_VEL
LIN {X 0,Y 216.336,Z 490.161,A -85,B 0,C 180,E1 -21842.628,E2 -21842.628} C_VEL
LIN {X 0,Y 220.659,Z 498.359,A -85,B 0,C 180,E1 -21845.25,E2 -21845.25} C_VEL
LIN {X 0,Y 226.828,Z 506.703,A -85,B 0,C 180,E1 -21848.356,E2 -21848.356} C_VEL
LIN {X 0,Y 234.876,Z 514.691,A -85,B 0,C 180,E1 -21851.806,E2 -21851.806} C_VEL
LIN {X 0,Y 243.21,Z 520.929,A -85,B 0,C 180,E1 -21854.926,E2 -21854.926} C_VEL
LIN {X 0,Y 251.569,Z 526.081,A -85,B 0,C 180,E1 -21857.895,E2 -21857.895} C_VEL
LIN {X 0,Y 259.318,Z 530.136,A -85,B 0,C 180,E1 -21860.642,E2 -21860.642} C_VEL
LIN {X 0,Y 263.86,Z 532.265,A -85,B 0,C 180,E1 -21862.347,E2 -21862.347} C_VEL
LIN {X 0,Y 268.392,Z 534.245,A -85,B 0,C 180,E1 -21864.288,E2 -21864.288} C_VEL
LIN {X 0,Y 270.582,Z 535.248,A -85,B 0,C 180,E1 -21865.531,E2 -21865.531} C_VEL
LIN {X 0,Y 274.25,Z 536.557,A -85,B 0,C 180,E1 -21868.024,E2 -21868.024} C_VEL
LIN {X 0,Y 276.168,Z 536.875,A -85,B 0,C 180,E1 -21870,E2 -21870} C_VEL
LIN {X 0,Y 274.25,Z 536.557,A -85,B 0,C 180,E1 -21871.975,E2 -21871.975} C_VEL
LIN {X 0,Y 270.566,Z 535.248,A -85,B 0,C 180,E1 -21874.469,E2 -21874.469} C_VEL
LIN {X 0,Y 267.63,Z 533.957,A -85,B 0,C 180,E1 -21876.029,E2 -21876.029} C_VEL
LIN {X 0,Y 262.657,Z 531.733,A -85,B 0,C 180,E1 -21878.108,E2 -21878.108} C_VEL
LIN {X 0,Y 257.045,Z 529.015,A -85,B 0,C 180,E1 -21880.173,E2 -21880.173} C_VEL
LIN {X 0,Y 248.85,Z 524.515,A -85,B 0,C 180,E1 -21883.058,E2 -21883.058} C_VEL
LIN {X 0,Y 241.072,Z 519.47,A -85,B 0,C 180,E1 -21885.839,E2 -21885.839} C_VEL
LIN {X 0,Y 233.701,Z 513.588,A -85,B 0,C 180,E1 -21888.692,E2 -21888.692} C_VEL
LIN {X 0,Y 226.317,Z 506.105,A -85,B 0,C 180,E1 -21891.878,E2 -21891.878} C_VEL
LIN {X 0,Y 220.708,Z 498.347,A -85,B 0,C 180,E1 -21894.747,E2 -21894.747} C_VEL
LIN {X 0,Y 216.331,Z 490.218,A -85,B 0,C 180,E1 -21897.359,E2 -21897.359} C_VEL
LIN {X 0,Y 212.835,Z 480.81,A -85,B 0,C 180,E1 -21899.914,E2 -21899.914} C_VEL
LIN {X 0,Y 209.61,Z 469.853,A -85,B 0,C 180,E1 -21902.442,E2 -21902.442} C_VEL
LIN {X 0,Y 204.952,Z 457.859,A -85,B 0,C 180,E1 -21905.048,E2 -21905.048} C_VEL
LIN {X 0,Y 200.134,Z 447.895,A -85,B 0,C 180,E1 -21907.186,E2 -21907.186} C_VEL
LIN {X 0,Y 195.954,Z 440.551,A -85,B 0,C 180,E1 -21908.817,E2 -21908.817} C_VEL
LIN {X 0,Y 194.468,Z 437.982,A -85,B 0,C 180,E1 -21909.364,E2 -21909.364} C_VEL
LIN {X 0,Y 192.922,Z 435.547,A -85,B 0,C 180,E1 -21909.911,E2 -21909.911} C_VEL
LIN {X 0,Y 192.549,Z 433.999,A -85,B 0,C 180,E1 -21910.126,E2 -21910.126} C_VEL
LIN {X 0,Y 192.509,Z 434.006,A -85,B 0,C 180,E1 -21913.918,E2 -21913.918} C_VEL
LIN {X 0,Y 192.509,Z 434.006,A -85,B 0,C 180,E1 -21918.92,E2 -21918.92} C_VEL
LIN {X 0,Y 192.581,Z 433.996,A -85,B 0,C 180,E1 -21923.403,E2 -21923.403} C_VEL
LIN {X 0,Y 192.605,Z 433.993,A -85,B 0,C 180,E1 -21927.059,E2 -21927.059} C_VEL
LIN {X 0,Y 192.66,Z 433.986,A -85,B 0,C 180,E1 -21931.693,E2 -21931.693} C_VEL
LIN {X 0,Y 192.701,Z 433.978,A -85,B 0,C 180,E1 -21936.349,E2 -21936.349} C_VEL
LIN {X 0,Y 192.727,Z 433.976,A -85,B 0,C 180,E1 -21941.459,E2 -21941.459} C_VEL
LIN {X 0,Y 192.76,Z 433.967,A -85,B 0,C 180,E1 -21945.215,E2 -21945.215} C_VEL
LIN {X 0,Y 192.941,Z 433.946,A -85,B 0,C 180,E1 -21949.568,E2 -21949.568} C_VEL
LIN {X 0,Y 192.981,Z 433.945,A -85,B 0,C 180,E1 -21953.729,E2 -21953.729} C_VEL
LIN {X 0,Y 193.258,Z 433.88,A -85,B 0,C 180,E1 -21957.917,E2 -21957.917} C_VEL
LIN {X 0,Y 193.439,Z 433.869,A -85,B 0,C 180,E1 -21960.001,E2 -21960.001} C_VEL
LIN {X 0,Y 192.97,Z 433.948,A -85,B 0,C 180,E1 -21964.178,E2 -21964.178} C_VEL
LIN {X 0,Y 193.033,Z 433.942,A -85,B 0,C 180,E1 -21968.375,E2 -21968.375} C_VEL
LIN {X 0,Y 192.798,Z 433.971,A -85,B 0,C 180,E1 -21972.635,E2 -21972.635} C_VEL
LIN {X 0,Y 192.753,Z 433.977,A -85,B 0,C 180,E1 -21976.96,E2 -21976.96} C_VEL
LIN {X 0,Y 192.619,Z 433.992,A -85,B 0,C 180,E1 -21981.4,E2 -21981.4} C_VEL
LIN {X 0,Y 192.646,Z 433.993,A -85,B 0,C 180,E1 -21984.214,E2 -21984.214} C_VEL
LIN {X 0,Y 192.842,Z 435.39,A -85,B 0,C 180,E1 -21988.997,E2 -21988.997} C_VEL
LIN {X 0,Y 193.003,Z 436.933,A -85,B 0,C 180,E1 -21993.123,E2 -21993.123} C_VEL
LIN {X 0,Y 193.261,Z 438.993,A -85,B 0,C 180,E1 -21998.187,E2 -21998.187} C_VEL
LIN {X 0,Y 193.46,Z 440.183,A -85,B 0,C 180,E1 -22000.838,E2 -22000.838} C_VEL
LIN {X 0,Y 193.546,Z 441.518,A -85,B 0,C 180,E1 -22003.625,E2 -22003.625} C_VEL
LIN {X 0,Y 193.472,Z 443.042,A -85,B 0,C 180,E1 -22006.596,E2 -22006.596} C_VEL
LIN {X 0,Y 193.103,Z 445.271,A -85,B 0,C 180,E1 -22010.254,E2 -22010.254} C_VEL
LIN {X 0,Y 194.127,Z 448.447,A -85,B 0,C 180,E1 -22010.708,E2 -22010.708} C_VEL
LIN {X 0,Y 195.244,Z 451.295,A -85,B 0,C 180,E1 -22011.226,E2 -22011.226} C_VEL
LIN {X 0,Y 198.827,Z 461.679,A -85,B 0,C 180,E1 -22013.066,E2 -22013.066} C_VEL
LIN {X 0,Y 201.325,Z 471.742,A -85,B 0,C 180,E1 -22014.874,E2 -22014.874} C_VEL
LIN {X 0,Y 203.101,Z 482.11,A -85,B 0,C 180,E1 -22016.862,E2 -22016.862} C_VEL
LIN {X 0,Y 203.836,Z 489.916,A -85,B 0,C 180,E1 -22018.45,E2 -22018.45} C_VEL
LIN {X 0,Y 204.18,Z 498.859,A -85,B 0,C 180,E1 -22020.468,E2 -22020.468} C_VEL
LIN {X 0,Y 203.883,Z 506.164,A -85,B 0,C 180,E1 -22022.267,E2 -22022.267} C_VEL
LIN {X 0,Y 200.999,Z 515.301,A -85,B 0,C 180,E1 -22024.639,E2 -22024.639} C_VEL
LIN {X 0,Y 198.876,Z 521.502,A -85,B 0,C 180,E1 -22026.575,E2 -22026.575} C_VEL
LIN {X 0,Y 196.717,Z 528.043,A -85,B 0,C 180,E1 -22029.068,E2 -22029.068} C_VEL
LIN {X 0,Y 195.103,Z 532.545,A -85,B 0,C 180,E1 -22031.083,E2 -22031.083} C_VEL
LIN {X 0,Y 193.06,Z 538.035,A -85,B 0,C 180,E1 -22034.156,E2 -22034.156} C_VEL
LIN {X 0,Y 191.672,Z 542.365,A -85,B 0,C 180,E1 -22037.291,E2 -22037.291} C_VEL
LIN {X 0,Y 191.031,Z 544.737,A -85,B 0,C 180,E1 -22039.4,E2 -22039.4} C_VEL
LIN {X 0,Y 190.545,Z 546.54,A -85,B 0,C 180,E1 -22041.516,E2 -22041.516} C_VEL
LIN {X 0,Y 190.166,Z 548.997,A -85,B 0,C 180,E1 -22045.761,E2 -22045.761} C_VEL
LIN {X 0,Y 190.153,Z 549.59,A -85,B 0,C 180,E1 -22047.882,E2 -22047.882} C_VEL
LIN {X 0,Y 190.248,Z 549.749,A -85,B 0,C 180,E1 -22050,E2 -22050} C_VEL
LIN {X 0,Y 190.121,Z 549.194,A -85,B 0,C 180,E1 -22053.534,E2 -22053.534} C_VEL
LIN {X 0,Y 190.282,Z 547.933,A -85,B 0,C 180,E1 -22056.362,E2 -22056.362} C_VEL
LIN {X 0,Y 190.545,Z 546.54,A -85,B 0,C 180,E1 -22058.484,E2 -22058.484} C_VEL
LIN {X 0,Y 191.231,Z 543.896,A -85,B 0,C 180,E1 -22061.371,E2 -22061.371} C_VEL
LIN {X 0,Y 191.128,Z 542.048,A -85,B 0,C 180,E1 -22063.046,E2 -22063.046} C_VEL
LIN {X 0,Y 189.523,Z 538.447,A -85,B 0,C 180,E1 -22065.791,E2 -22065.791} C_VEL
LIN {X 0,Y 188.258,Z 534.314,A -85,B 0,C 180,E1 -22068.5,E2 -22068.5} C_VEL
LIN {X 0,Y 188.684,Z 531.462,A -85,B 0,C 180,E1 -22070.07,E2 -22070.07} C_VEL
LIN {X 0,Y 191.302,Z 524.492,A -85,B 0,C 180,E1 -22073.081,E2 -22073.081} C_VEL
LIN {X 0,Y 193.371,Z 518.355,A -85,B 0,C 180,E1 -22075.28,E2 -22075.28} C_VEL
LIN {X 0,Y 196.387,Z 509.806,A -85,B 0,C 180,E1 -22077.724,E2 -22077.724} C_VEL
LIN {X 0,Y 197.318,Z 505.957,A -85,B 0,C 180,E1 -22078.739,E2 -22078.739} C_VEL
LIN {X 0,Y 197.644,Z 495.365,A -85,B 0,C 180,E1 -22081.413,E2 -22081.413} C_VEL
LIN {X 0,Y 197.04,Z 486.021,A -85,B 0,C 180,E1 -22083.527,E2 -22083.527} C_VEL
LIN {X 0,Y 195.579,Z 475.809,A -85,B 0,C 180,E1 -22085.65,E2 -22085.65} C_VEL
LIN {X 0,Y 193.583,Z 466.341,A -85,B 0,C 180,E1 -22087.494,E2 -22087.494} C_VEL
LIN {X 0,Y 190.19,Z 455.657,A -85,B 0,C 180,E1 -22089.563,E2 -22089.563} C_VEL
LIN {X 0,Y 187.608,Z 448.868,A -85,B 0,C 180,E1 -22090.886,E2 -22090.886} C_VEL
LIN {X 0,Y 186.325,Z 445.77,A -85,B 0,C 180,E1 -22091.45,E2 -22091.45} C_VEL
LIN {X 0,Y 186.2,Z 444.812,A -85,B 0,C 180,E1 -22091.625,E2 -22091.625} C_VEL
LIN {X 0,Y 186.464,Z 442.702,A -85,B 0,C 180,E1 -22095.734,E2 -22095.734} C_VEL
LIN {X 0,Y 186.362,Z 440.682,A -85,B 0,C 180,E1 -22100.125,E2 -22100.125} C_VEL
LIN {X 0,Y 186.015,Z 438.475,A -85,B 0,C 180,E1 -22105.476,E2 -22105.476} C_VEL
LIN {X 0,Y 185.831,Z 436.641,A -85,B 0,C 180,E1 -22110.549,E2 -22110.549} C_VEL
LIN {X 0,Y 185.623,Z 435.098,A -85,B 0,C 180,E1 -22115.386,E2 -22115.386} C_VEL
LIN {X 0,Y 185.599,Z 434.868,A -85,B 0,C 180,E1 -22120.073,E2 -22120.073} C_VEL
LIN {X 0,Y 185.69,Z 434.855,A -85,B 0,C 180,E1 -22124.636,E2 -22124.636} C_VEL
LIN {X 0,Y 185.886,Z 434.831,A -85,B 0,C 180,E1 -22129.417,E2 -22129.417} C_VEL
LIN {X 0,Y 185.944,Z 434.824,A -85,B 0,C 180,E1 -22133.488,E2 -22133.488} C_VEL
LIN {X 0,Y 186.203,Z 434.787,A -85,B 0,C 180,E1 -22137.836,E2 -22137.836} C_VEL
LIN {X 0,Y 186.402,Z 434.743,A -85,B 0,C 180,E1 -22139.999,E2 -22139.999} C_VEL
LIN {X 0,Y 185.916,Z 434.811,A -85,B 0,C 180,E1 -22144.335,E2 -22144.335} C_VEL
LIN {X 0,Y 185.982,Z 434.814,A -85,B 0,C 180,E1 -22148.693,E2 -22148.693} C_VEL
LIN {X 0,Y 185.725,Z 434.849,A -85,B 0,C 180,E1 -22153.122,E2 -22153.122} C_VEL
LIN {X 0,Y 185.686,Z 434.855,A -85,B 0,C 180,E1 -22157.624,E2 -22157.624} C_VEL
LIN {X 0,Y 185.592,Z 434.867,A -85,B 0,C 180,E1 -22162.251,E2 -22162.251} C_VEL
LIN {X 0,Y 185.558,Z 434.872,A -85,B 0,C 180,E1 -22167.031,E2 -22167.031} C_VEL
LIN {X 0,Y 185.575,Z 434.87,A -85,B 0,C 180,E1 -22169.492,E2 -22169.492} C_VEL
LIN {X 0,Y 185.516,Z 434.877,A -85,B 0,C 180,E1 -22174.627,E2 -22174.627} C_VEL
LIN {X 0,Y 185.563,Z 434.87,A -85,B 0,C 180,E1 -22177.313,E2 -22177.313} C_VEL
LIN {X 0,Y 185.567,Z 434.869,A -85,B 0,C 180,E1 -22180.76,E2 -22180.76} C_VEL
LIN {X 0,Y 185.55,Z 434.873,A -85,B 0,C 180,E1 -22183.975,E2 -22183.975} C_VEL
LIN {X 0,Y 185.481,Z 434.992,A -85,B 0,C 180,E1 -22188.11,E2 -22188.11} C_VEL
LIN {X 0,Y 186.525,Z 437.811,A -85,B 0,C 180,E1 -22188.591,E2 -22188.591} C_VEL
LIN {X 0,Y 188.259,Z 439.987,A -85,B 0,C 180,E1 -22189.205,E2 -22189.205} C_VEL
LIN {X 0,Y 194.445,Z 450.932,A -85,B 0,C 180,E1 -22191.823,E2 -22191.823} C_VEL
LIN {X 0,Y 199.237,Z 461.236,A -85,B 0,C 180,E1 -22194.222,E2 -22194.222} C_VEL
LIN {X 0,Y 203.049,Z 471.422,A -85,B 0,C 180,E1 -22196.616,E2 -22196.616} C_VEL
LIN {X 0,Y 205.562,Z 480.172,A -85,B 0,C 180,E1 -22198.728,E2 -22198.728} C_VEL
LIN {X 0,Y 208.166,Z 488.732,A -85,B 0,C 180,E1 -22201.044,E2 -22201.044} C_VEL
LIN {X 0,Y 211.736,Z 496.939,A -85,B 0,C 180,E1 -22203.659,E2 -22203.659} C_VEL
LIN {X 0,Y 216.524,Z 504.749,A -85,B 0,C 180,E1 -22206.558,E2 -22206.558} C_VEL
LIN {X 0,Y 221.586,Z 510.858,A -85,B 0,C 180,E1 -22209.139,E2 -22209.139} C_VEL
LIN {X 0,Y 228.674,Z 517.468,A -85,B 0,C 180,E1 -22212.312,E2 -22212.312} C_VEL
LIN {X 0,Y 236.202,Z 522.781,A -85,B 0,C 180,E1 -22215.234,E2 -22215.234} C_VEL
LIN {X 0,Y 244.975,Z 527.806,A -85,B 0,C 180,E1 -22218.415,E2 -22218.415} C_VEL
LIN {X 0,Y 252.748,Z 531.491,A -85,B 0,C 180,E1 -22221.203,E2 -22221.203} C_VEL
LIN {X 0,Y 259.316,Z 534.19,A -85,B 0,C 180,E1 -22223.777,E2 -22223.777} C_VEL
LIN {X 0,Y 262.786,Z 535.463,A -85,B 0,C 180,E1 -22225.398,E2 -22225.398} C_VEL
LIN {X 0,Y 265.268,Z 536.399,A -85,B 0,C 180,E1 -22226.963,E2 -22226.963} C_VEL
LIN {X 0,Y 267.516,Z 536.921,A -85,B 0,C 180,E1 -22228.495,E2 -22228.495} C_VEL
LIN {X 0,Y 268.94,Z 537.072,A -85,B 0,C 180,E1 -22230,E2 -22230} C_VEL
LIN {X 0,Y 267.183,Z 536.85,A -85,B 0,C 180,E1 -22231.74,E2 -22231.74} C_VEL
LIN {X 0,Y 265.263,Z 536.398,A -85,B 0,C 180,E1 -22233.037,E2 -22233.037} C_VEL
LIN {X 0,Y 262.753,Z 535.464,A -85,B 0,C 180,E1 -22234.602,E2 -22234.602} C_VEL
LIN {X 0,Y 259.283,Z 534.191,A -85,B 0,C 180,E1 -22236.224,E2 -22236.224} C_VEL
LIN {X 0,Y 255.102,Z 532.51,A -85,B 0,C 180,E1 -22237.917,E2 -22237.917} C_VEL
LIN {X 0,Y 247.654,Z 529.171,A -85,B 0,C 180,E1 -22240.632,E2 -22240.632} C_VEL
LIN {X 0,Y 238.803,Z 524.457,A -85,B 0,C 180,E1 -22243.79,E2 -22243.79} C_VEL
LIN {X 0,Y 231.149,Z 519.324,A -85,B 0,C 180,E1 -22246.719,E2 -22246.719} C_VEL
LIN {X 0,Y 222.757,Z 512.056,A -85,B 0,C 180,E1 -22250.307,E2 -22250.307} C_VEL
LIN {X 0,Y 217.757,Z 506.355,A -85,B 0,C 180,E1 -22252.786,E2 -22252.786} C_VEL
LIN {X 0,Y 212.866,Z 498.959,A -85,B 0,C 180,E1 -22255.619,E2 -22255.619} C_VEL
LIN {X 0,Y 209.304,Z 491.743,A -85,B 0,C 180,E1 -22258.039,E2 -22258.039} C_VEL
LIN {X 0,Y 206.508,Z 483.589,A -85,B 0,C 180,E1 -22260.381,E2 -22260.381} C_VEL
LIN {X 0,Y 203.807,Z 473.8,A -85,B 0,C 180,E1 -22262.805,E2 -22262.805} C_VEL
LIN {X 0,Y 200.973,Z 465.652,A -85,B 0,C 180,E1 -22264.736,E2 -22264.736} C_VEL
LIN {X 0,Y 197.359,Z 456.926,A -85,B 0,C 180,E1 -22266.756,E2 -22266.756} C_VEL
LIN {X 0,Y 192.226,Z 446.815,A -85,B 0,C 180,E1 -22269.126,E2 -22269.126} C_VEL
LIN {X 0,Y 188.247,Z 440.037,A -85,B 0,C 180,E1 -22270.794,E2 -22270.794} C_VEL
LIN {X 0,Y 185.933,Z 436.693,A -85,B 0,C 180,E1 -22271.672,E2 -22271.672} C_VEL
LIN {X 0,Y 185.453,Z 434.884,A -85,B 0,C 180,E1 -22271.97,E2 -22271.97} C_VEL
LIN {X 0,Y 185.453,Z 434.883,A -85,B 0,C 180,E1 -22276.991,E2 -22276.991} C_VEL
LIN {X 0,Y 185.463,Z 434.882,A -85,B 0,C 180,E1 -22279.896,E2 -22279.896} C_VEL
LIN {X 0,Y 185.501,Z 434.878,A -85,B 0,C 180,E1 -22282.712,E2 -22282.712} C_VEL
LIN {X 0,Y 185.541,Z 434.873,A -85,B 0,C 180,E1 -22287.976,E2 -22287.976} C_VEL
LIN {X 0,Y 185.577,Z 434.87,A -85,B 0,C 180,E1 -22290.576,E2 -22290.576} C_VEL
LIN {X 0,Y 185.583,Z 434.861,A -85,B 0,C 180,E1 -22295.383,E2 -22295.383} C_VEL
LIN {X 0,Y 185.67,Z 434.852,A -85,B 0,C 180,E1 -22301.134,E2 -22301.134} C_VEL
LIN {X 0,Y 185.691,Z 434.848,A -85,B 0,C 180,E1 -22304.638,E2 -22304.638} C_VEL
LIN {X 0,Y 185.885,Z 434.826,A -85,B 0,C 180,E1 -22309.419,E2 -22309.419} C_VEL
LIN {X 0,Y 185.943,Z 434.822,A -85,B 0,C 180,E1 -22313.491,E2 -22313.491} C_VEL
LIN {X 0,Y 186.202,Z 434.757,A -85,B 0,C 180,E1 -22317.838,E2 -22317.838} C_VEL
LIN {X 0,Y 186.402,Z 434.743,A -85,B 0,C 180,E1 -22320.001,E2 -22320.001} C_VEL
LIN {X 0,Y 185.917,Z 434.827,A -85,B 0,C 180,E1 -22324.337,E2 -22324.337} C_VEL
LIN {X 0,Y 185.98,Z 434.819,A -85,B 0,C 180,E1 -22328.695,E2 -22328.695} C_VEL
LIN {X 0,Y 185.725,Z 434.852,A -85,B 0,C 180,E1 -22333.124,E2 -22333.124} C_VEL
LIN {X 0,Y 185.687,Z 434.857,A -85,B 0,C 180,E1 -22337.626,E2 -22337.626} C_VEL
LIN {X 0,Y 185.579,Z 434.871,A -85,B 0,C 180,E1 -22342.255,E2 -22342.255} C_VEL
LIN {X 0,Y 185.616,Z 435.12,A -85,B 0,C 180,E1 -22344.675,E2 -22344.675} C_VEL
LIN {X 0,Y 185.831,Z 436.681,A -85,B 0,C 180,E1 -22349.562,E2 -22349.562} C_VEL
LIN {X 0,Y 186.015,Z 438.474,A -85,B 0,C 180,E1 -22354.524,E2 -22354.524} C_VEL
LIN {X 0,Y 186.364,Z 440.68,A -85,B 0,C 180,E1 -22359.875,E2 -22359.875} C_VEL
LIN {X 0,Y 186.462,Z 442.701,A -85,B 0,C 180,E1 -22364.265,E2 -22364.265} C_VEL
LIN {X 0,Y 186.18,Z 444.901,A -85,B 0,C 180,E1 -22368.449,E2 -22368.449} C_VEL
LIN {X 0,Y 187.088,Z 447.941,A -85,B 0,C 180,E1 -22368.902,E2 -22368.902} C_VEL
LIN {X 0,Y 188.229,Z 450.251,A -85,B 0,C 180,E1 -22369.41,E2 -22369.41} C_VEL
LIN {X 0,Y 191.63,Z 459.663,A -85,B 0,C 180,E1 -22371.202,E2 -22371.202} C_VEL
LIN {X 0,Y 194.426,Z 469.711,A -85,B 0,C 180,E1 -22373.146,E2 -22373.146} C_VEL
LIN {X 0,Y 196.412,Z 480.869,A -85,B 0,C 180,E1 -22375.386,E2 -22375.386} C_VEL
LIN {X 0,Y 197.351,Z 489.997,A -85,B 0,C 180,E1 -22377.352,E2 -22377.352} C_VEL
LIN {X 0,Y 197.654,Z 499.235,A -85,B 0,C 180,E1 -22379.542,E2 -22379.542} C_VEL
LIN {X 0,Y 197.348,Z 505.958,A -85,B 0,C 180,E1 -22381.265,E2 -22381.265} C_VEL
LIN {X 0,Y 196.403,Z 509.807,A -85,B 0,C 180,E1 -22382.278,E2 -22382.278} C_VEL
LIN {X 0,Y 193.447,Z 518.357,A -85,B 0,C 180,E1 -22384.731,E2 -22384.731} C_VEL
LIN {X 0,Y 190.504,Z 526.822,A -85,B 0,C 180,E1 -22387.847,E2 -22387.847} C_VEL
LIN {X 0,Y 188.355,Z 532.346,A -85,B 0,C 180,E1 -22390.379,E2 -22390.379} C_VEL
LIN {X 0,Y 186.212,Z 537.838,A -85,B 0,C 180,E1 -22393.557,E2 -22393.557} C_VEL
LIN {X 0,Y 184.729,Z 542.168,A -85,B 0,C 180,E1 -22396.805,E2 -22396.805} C_VEL
LIN {X 0,Y 184.039,Z 544.539,A -85,B 0,C 180,E1 -22398.993,E2 -22398.993} C_VEL
LIN {X 0,Y 183.515,Z 546.342,A -85,B 0,C 180,E1 -22401.189,E2 -22401.189} C_VEL
LIN {X 0,Y 183.08,Z 548.799,A -85,B 0,C 180,E1 -22405.597,E2 -22405.597} C_VEL
LIN {X 0,Y 183.052,Z 549.393,A -85,B 0,C 180,E1 -22407.8,E2 -22407.8} C_VEL
LIN {X 0,Y 183.154,Z 549.552,A -85,B 0,C 180,E1 -22410,E2 -22410} C_VEL
LIN {X 0,Y 183.02,Z 549.119,A -85,B 0,C 180,E1 -22413.217,E2 -22413.217} C_VEL
LIN {X 0,Y 183.215,Z 547.735,A -85,B 0,C 180,E1 -22416.608,E2 -22416.608} C_VEL
LIN {X 0,Y 183.515,Z 546.342,A -85,B 0,C 180,E1 -22418.811,E2 -22418.811} C_VEL
LIN {X 0,Y 184.343,Z 543.386,A -85,B 0,C 180,E1 -22422.104,E2 -22422.104} C_VEL
LIN {X 0,Y 185.603,Z 539.391,A -85,B 0,C 180,E1 -22425.37,E2 -22425.37} C_VEL
LIN {X 0,Y 187.609,Z 534.263,A -85,B 0,C 180,E1 -22428.567,E2 -22428.567} C_VEL
LIN {X 0,Y 188.684,Z 531.462,A -85,B 0,C 180,E1 -22430.07,E2 -22430.07} C_VEL
LIN {X 0,Y 189.19,Z 528.4,A -85,B 0,C 180,E1 -22431.597,E2 -22431.597} C_VEL
LIN {X 0,Y 188.489,Z 523.014,A -85,B 0,C 180,E1 -22434.12,E2 -22434.12} C_VEL
LIN {X 0,Y 188.04,Z 517.018,A -85,B 0,C 180,E1 -22436.518,E2 -22436.518} C_VEL
LIN {X 0,Y 188.905,Z 513.003,A -85,B 0,C 180,E1 -22437.807,E2 -22437.807} C_VEL
LIN {X 0,Y 190.597,Z 507.684,A -85,B 0,C 180,E1 -22439.246,E2 -22439.246} C_VEL
LIN {X 0,Y 191.128,Z 500.186,A -85,B 0,C 180,E1 -22441.303,E2 -22441.303} C_VEL
LIN {X 0,Y 191.025,Z 492.709,A -85,B 0,C 180,E1 -22443.195,E2 -22443.195} C_VEL
LIN {X 0,Y 190.365,Z 484.068,A -85,B 0,C 180,E1 -22445.208,E2 -22445.208} C_VEL
LIN {X 0,Y 188.989,Z 474.864,A -85,B 0,C 180,E1 -22447.215,E2 -22447.215} C_VEL
LIN {X 0,Y 186.883,Z 465.732,A -85,B 0,C 180,E1 -22449.137,E2 -22449.137} C_VEL
LIN {X 0,Y 183.595,Z 455.483,A -85,B 0,C 180,E1 -22451.278,E2 -22451.278} C_VEL
LIN {X 0,Y 181.047,Z 449.121,A -85,B 0,C 180,E1 -22452.659,E2 -22452.659} C_VEL
LIN {X 0,Y 179.565,Z 446.031,A -85,B 0,C 180,E1 -22453.346,E2 -22453.346} C_VEL
LIN {X 0,Y 179.315,Z 444.601,A -85,B 0,C 180,E1 -22453.559,E2 -22453.559} C_VEL
LIN {X 0,Y 179.371,Z 442.443,A -85,B 0,C 180,E1 -22458.233,E2 -22458.233} C_VEL
LIN {X 0,Y 179.194,Z 440.988,A -85,B 0,C 180,E1 -22461.664,E2 -22461.664} C_VEL
LIN {X 0,Y 178.921,Z 439.045,A -85,B 0,C 180,E1 -22466.637,E2 -22466.637} C_VEL
LIN {X 0,Y 178.715,Z 437.283,A -85,B 0,C 180,E1 -22471.841,E2 -22471.841} C_VEL
LIN {X 0,Y 178.512,Z 435.82,A -85,B 0,C 180,E1 -22476.814,E2 -22476.814} C_VEL
LIN {X 0,Y 178.647,Z 435.734,A -85,B 0,C 180,E1 -22481.655,E2 -22481.655} C_VEL
LIN {X 0,Y 178.654,Z 435.732,A -85,B 0,C 180,E1 -22486.346,E2 -22486.346} C_VEL
LIN {X 0,Y 178.908,Z 435.699,A -85,B 0,C 180,E1 -22490.958,E2 -22490.958} C_VEL
LIN {X 0,Y 179.149,Z 435.666,A -85,B 0,C 180,E1 -22497.75,E2 -22497.75} C_VEL
LIN {X 0,Y 179.366,Z 435.618,A -85,B 0,C 180,E1 -22499.999,E2 -22499.999} C_VEL
LIN {X 0,Y 178.864,Z 435.691,A -85,B 0,C 180,E1 -22504.506,E2 -22504.506} C_VEL
LIN {X 0,Y 178.91,Z 435.692,A -85,B 0,C 180,E1 -22509.039,E2 -22509.039} C_VEL
LIN {X 0,Y 178.653,Z 435.726,A -85,B 0,C 180,E1 -22513.651,E2 -22513.651} C_VEL
LIN {X 0,Y 178.619,Z 435.728,A -85,B 0,C 180,E1 -22519.215,E2 -22519.215} C_VEL
LIN {X 0,Y 178.52,Z 435.74,A -85,B 0,C 180,E1 -22525.117,E2 -22525.117} C_VEL
LIN {X 0,Y 178.518,Z 435.748,A -85,B 0,C 180,E1 -22529.993,E2 -22529.993} C_VEL
LIN {X 0,Y 178.48,Z 435.752,A -85,B 0,C 180,E1 -22534.219,E2 -22534.219} C_VEL
LIN {X 0,Y 178.476,Z 435.754,A -85,B 0,C 180,E1 -22539.052,E2 -22539.052} C_VEL
LIN {X 0,Y 178.496,Z 435.751,A -85,B 0,C 180,E1 -22542.015,E2 -22542.015} C_VEL
LIN {X 0,Y 178.467,Z 435.795,A -85,B 0,C 180,E1 -22546.096,E2 -22546.096} C_VEL
LIN {X 0,Y 179.382,Z 438.475,A -85,B 0,C 180,E1 -22546.575,E2 -22546.575} C_VEL
LIN {X 0,Y 181.323,Z 440.959,A -85,B 0,C 180,E1 -22547.346,E2 -22547.346} C_VEL
LIN {X 0,Y 183.173,Z 444.155,A -85,B 0,C 180,E1 -22548.216,E2 -22548.216} C_VEL
LIN {X 0,Y 187.705,Z 452.024,A -85,B 0,C 180,E1 -22550.3,E2 -22550.3} C_VEL
LIN {X 0,Y 192.533,Z 462.261,A -85,B 0,C 180,E1 -22552.903,E2 -22552.903} C_VEL
LIN {X 0,Y 196.309,Z 472.24,A -85,B 0,C 180,E1 -22555.426,E2 -22555.426} C_VEL
LIN {X 0,Y 199.054,Z 481.901,A -85,B 0,C 180,E1 -22557.924,E2 -22557.924} C_VEL
LIN {X 0,Y 201.267,Z 490.189,A -85,B 0,C 180,E1 -22560.272,E2 -22560.272} C_VEL
LIN {X 0,Y 204.264,Z 497.775,A -85,B 0,C 180,E1 -22562.796,E2 -22562.796} C_VEL
LIN {X 0,Y 208.31,Z 505.162,A -85,B 0,C 180,E1 -22565.631,E2 -22565.631} C_VEL
LIN {X 0,Y 213.878,Z 512.313,A -85,B 0,C 180,E1 -22568.811,E2 -22568.811} C_VEL
LIN {X 0,Y 221.279,Z 519.166,A -85,B 0,C 180,E1 -22572.327,E2 -22572.327} C_VEL
LIN {X 0,Y 229.947,Z 525.058,A -85,B 0,C 180,E1 -22575.848,E2 -22575.848} C_VEL
LIN {X 0,Y 236.759,Z 528.709,A -85,B 0,C 180,E1 -22578.395,E2 -22578.395} C_VEL
LIN {X 0,Y 242.338,Z 531.206,A -85,B 0,C 180,E1 -22580.405,E2 -22580.405} C_VEL
LIN {X 0,Y 248.095,Z 533.461,A -85,B 0,C 180,E1 -22582.506,E2 -22582.506} C_VEL
LIN {X 0,Y 254.814,Z 535.684,A -85,B 0,C 180,E1 -22585.254,E2 -22585.254} C_VEL
LIN {X 0,Y 257.63,Z 536.612,A -85,B 0,C 180,E1 -22586.873,E2 -22586.873} C_VEL
LIN {X 0,Y 260.119,Z 537.146,A -85,B 0,C 180,E1 -22588.514,E2 -22588.514} C_VEL
LIN {X 0,Y 261.681,Z 537.269,A -85,B 0,C 180,E1 -22590,E2 -22590} C_VEL
LIN {X 0,Y 260.033,Z 537.128,A -85,B 0,C 180,E1 -22591.549,E2 -22591.549} C_VEL
LIN {X 0,Y 257.615,Z 536.612,A -85,B 0,C 180,E1 -22593.128,E2 -22593.128} C_VEL
LIN {X 0,Y 254.005,Z 535.457,A -85,B 0,C 180,E1 -22595.091,E2 -22595.091} C_VEL
LIN {X 0,Y 248.095,Z 533.46,A -85,B 0,C 180,E1 -22597.495,E2 -22597.495} C_VEL
LIN {X 0,Y 241.012,Z 530.642,A -85,B 0,C 180,E1 -22600.076,E2 -22600.076} C_VEL
LIN {X 0,Y 231.368,Z 525.919,A -85,B 0,C 180,E1 -22603.589,E2 -22603.589} C_VEL
LIN {X 0,Y 223.458,Z 520.811,A -85,B 0,C 180,E1 -22606.755,E2 -22606.755} C_VEL
LIN {X 0,Y 216.645,Z 515.134,A -85,B 0,C 180,E1 -22609.823,E2 -22609.823} C_VEL
LIN {X 0,Y 210.284,Z 507.898,A -85,B 0,C 180,E1 -22613.212,E2 -22613.212} C_VEL
LIN {X 0,Y 205.313,Z 499.915,A -85,B 0,C 180,E1 -22616.423,E2 -22616.423} C_VEL
LIN {X 0,Y 202.419,Z 493.222,A -85,B 0,C 180,E1 -22618.76,E2 -22618.76} C_VEL
LIN {X 0,Y 199.673,Z 484.396,A -85,B 0,C 180,E1 -22621.406,E2 -22621.406} C_VEL
LIN {X 0,Y 197.179,Z 474.962,A -85,B 0,C 180,E1 -22623.874,E2 -22623.874} C_VEL
LIN {X 0,Y 193.875,Z 465.659,A -85,B 0,C 180,E1 -22626.24,E2 -22626.24} C_VEL
LIN {X 0,Y 190.054,Z 456.852,A -85,B 0,C 180,E1 -22628.461,E2 -22628.461} C_VEL
LIN {X 0,Y 185.116,Z 447.521,A -85,B 0,C 180,E1 -22630.892,E2 -22630.892} C_VEL
LIN {X 0,Y 182.762,Z 443.677,A -85,B 0,C 180,E1 -22631.951,E2 -22631.951} C_VEL
LIN {X 0,Y 180.66,Z 440.101,A -85,B 0,C 180,E1 -22632.923,E2 -22632.923} C_VEL
LIN {X 0,Y 178.986,Z 437.768,A -85,B 0,C 180,E1 -22633.619,E2 -22633.619} C_VEL
LIN {X 0,Y 178.435,Z 435.759,A -85,B 0,C 180,E1 -22633.995,E2 -22633.995} C_VEL
LIN {X 0,Y 178.399,Z 435.763,A -85,B 0,C 180,E1 -22638.459,E2 -22638.459} C_VEL
LIN {X 0,Y 178.418,Z 435.759,A -85,B 0,C 180,E1 -22643.784,E2 -22643.784} C_VEL
LIN {X 0,Y 178.482,Z 435.751,A -85,B 0,C 180,E1 -22646.547,E2 -22646.547} C_VEL
LIN {X 0,Y 178.518,Z 435.748,A -85,B 0,C 180,E1 -22650.007,E2 -22650.007} C_VEL
LIN {X 0,Y 178.52,Z 435.74,A -85,B 0,C 180,E1 -22654.883,E2 -22654.883} C_VEL
LIN {X 0,Y 178.619,Z 435.728,A -85,B 0,C 180,E1 -22660.785,E2 -22660.785} C_VEL
LIN {X 0,Y 178.653,Z 435.726,A -85,B 0,C 180,E1 -22666.349,E2 -22666.349} C_VEL
LIN {X 0,Y 178.907,Z 435.693,A -85,B 0,C 180,E1 -22670.961,E2 -22670.961} C_VEL
LIN {X 0,Y 178.862,Z 435.691,A -85,B 0,C 180,E1 -22675.494,E2 -22675.494} C_VEL
LIN {X 0,Y 179.366,Z 435.618,A -85,B 0,C 180,E1 -22680.001,E2 -22680.001} C_VEL
LIN {X 0,Y 178.864,Z 435.705,A -85,B 0,C 180,E1 -22684.508,E2 -22684.508} C_VEL
LIN {X 0,Y 178.908,Z 435.7,A -85,B 0,C 180,E1 -22689.042,E2 -22689.042} C_VEL
LIN {X 0,Y 178.654,Z 435.733,A -85,B 0,C 180,E1 -22693.654,E2 -22693.654} C_VEL
LIN {X 0,Y 178.62,Z 435.736,A -85,B 0,C 180,E1 -22699.216,E2 -22699.216} C_VEL
LIN {X 0,Y 178.512,Z 435.821,A -85,B 0,C 180,E1 -22703.186,E2 -22703.186} C_VEL
LIN {X 0,Y 178.715,Z 437.282,A -85,B 0,C 180,E1 -22708.159,E2 -22708.159} C_VEL
LIN {X 0,Y 178.921,Z 439.042,A -85,B 0,C 180,E1 -22713.363,E2 -22713.363} C_VEL
LIN {X 0,Y 179.228,Z 441.202,A -85,B 0,C 180,E1 -22718.86,E2 -22718.86} C_VEL
LIN {X 0,Y 179.383,Z 442.497,A -85,B 0,C 180,E1 -22721.894,E2 -22721.894} C_VEL
LIN {X 0,Y 179.301,Z 444.638,A -85,B 0,C 180,E1 -22726.446,E2 -22726.446} C_VEL
LIN {X 0,Y 180.282,Z 447.843,A -85,B 0,C 180,E1 -22726.999,E2 -22726.999} C_VEL
LIN {X 0,Y 181.468,Z 450.129,A -85,B 0,C 180,E1 -22727.569,E2 -22727.569} C_VEL
LIN {X 0,Y 184.925,Z 459.139,A -85,B 0,C 180,E1 -22729.474,E2 -22729.474} C_VEL
LIN {X 0,Y 188.204,Z 470.802,A -85,B 0,C 180,E1 -22731.932,E2 -22731.932} C_VEL
LIN {X 0,Y 189.925,Z 480.655,A -85,B 0,C 180,E1 -22734.026,E2 -22734.026} C_VEL
LIN {X 0,Y 190.931,Z 490.082,A -85,B 0,C 180,E1 -22736.179,E2 -22736.179} C_VEL
LIN {X 0,Y 191.179,Z 499.002,A -85,B 0,C 180,E1 -22738.387,E2 -22738.387} C_VEL
LIN {X 0,Y 190.873,Z 505.752,A -85,B 0,C 180,E1 -22740.194,E2 -22740.194} C_VEL
LIN {X 0,Y 190.128,Z 509.609,A -85,B 0,C 180,E1 -22741.28,E2 -22741.28} C_VEL
LIN {X 0,Y 187.016,Z 518.159,A -85,B 0,C 180,E1 -22743.797,E2 -22743.797} C_VEL
LIN {X 0,Y 184.036,Z 526.341,A -85,B 0,C 180,E1 -22746.879,E2 -22746.879} C_VEL
LIN {X 0,Y 181.632,Z 532.148,A -85,B 0,C 180,E1 -22749.621,E2 -22749.621} C_VEL
LIN {X 0,Y 179.392,Z 537.64,A -85,B 0,C 180,E1 -22752.913,E2 -22752.913} C_VEL
LIN {X 0,Y 177.785,Z 541.969,A -85,B 0,C 180,E1 -22756.28,E2 -22756.28} C_VEL
LIN {X 0,Y 177.035,Z 544.341,A -85,B 0,C 180,E1 -22758.552,E2 -22758.552} C_VEL
LIN {X 0,Y 176.477,Z 546.145,A -85,B 0,C 180,E1 -22760.834,E2 -22760.834} C_VEL
LIN {X 0,Y 176.01,Z 548.603,A -85,B 0,C 180,E1 -22765.42,E2 -22765.42} C_VEL
LIN {X 0,Y 175.972,Z 549.196,A -85,B 0,C 180,E1 -22767.711,E2 -22767.711} C_VEL
LIN {X 0,Y 176.062,Z 549.355,A -85,B 0,C 180,E1 -22770,E2 -22770} C_VEL
LIN {X 0,Y 175.951,Z 549.003,A -85,B 0,C 180,E1 -22773.037,E2 -22773.037} C_VEL
LIN {X 0,Y 176.143,Z 547.538,A -85,B 0,C 180,E1 -22776.875,E2 -22776.875} C_VEL
LIN {X 0,Y 176.477,Z 546.145,A -85,B 0,C 180,E1 -22779.166,E2 -22779.166} C_VEL
LIN {X 0,Y 177.392,Z 543.189,A -85,B 0,C 180,E1 -22782.585,E2 -22782.585} C_VEL
LIN {X 0,Y 178.733,Z 539.193,A -85,B 0,C 180,E1 -22785.976,E2 -22785.976} C_VEL
LIN {X 0,Y 180.869,Z 534.065,A -85,B 0,C 180,E1 -22789.286,E2 -22789.286} C_VEL
LIN {X 0,Y 183.009,Z 528.803,A -85,B 0,C 180,E1 -22791.988,E2 -22791.988} C_VEL
LIN {X 0,Y 185.364,Z 522.483,A -85,B 0,C 180,E1 -22794.649,E2 -22794.649} C_VEL
LIN {X 0,Y 187.561,Z 516.531,A -85,B 0,C 180,E1 -22796.72,E2 -22796.72} C_VEL
LIN {X 0,Y 188.905,Z 513.003,A -85,B 0,C 180,E1 -22797.807,E2 -22797.807} C_VEL
LIN {X 0,Y 189.485,Z 510.257,A -85,B 0,C 180,E1 -22798.632,E2 -22798.632} C_VEL
LIN {X 0,Y 189.11,Z 506.27,A -85,B 0,C 180,E1 -22799.948,E2 -22799.948} C_VEL
LIN {X 0,Y 187.844,Z 502.441,A -85,B 0,C 180,E1 -22801.29,E2 -22801.29} C_VEL
LIN {X 0,Y 185.751,Z 497.209,A -85,B 0,C 180,E1 -22803.103,E2 -22803.103} C_VEL
LIN {X 0,Y 184.715,Z 492.858,A -85,B 0,C 180,E1 -22804.4,E2 -22804.4} C_VEL
LIN {X 0,Y 184.568,Z 491.298,A -85,B 0,C 180,E1 -22804.807,E2 -22804.807} C_VEL
LIN {X 0,Y 183.935,Z 483.821,A -85,B 0,C 180,E1 -22806.639,E2 -22806.639} C_VEL
LIN {X 0,Y 182.808,Z 475.79,A -85,B 0,C 180,E1 -22808.502,E2 -22808.502} C_VEL
LIN {X 0,Y 180.274,Z 464.963,A -85,B 0,C 180,E1 -22810.943,E2 -22810.943} C_VEL
LIN {X 0,Y 177.344,Z 456.382,A -85,B 0,C 180,E1 -22812.951,E2 -22812.951} C_VEL
LIN {X 0,Y 175.626,Z 452.371,A -85,B 0,C 180,E1 -22813.919,E2 -22813.919} C_VEL
LIN {X 0,Y 174.251,Z 448.997,A -85,B 0,C 180,E1 -22814.739,E2 -22814.739} C_VEL
LIN {X 0,Y 172.662,Z 446.014,A -85,B 0,C 180,E1 -22815.53,E2 -22815.53} C_VEL
LIN {X 0,Y 172.311,Z 444.335,A -85,B 0,C 180,E1 -22815.852,E2 -22815.852} C_VEL
LIN {X 0,Y 172.194,Z 442.263,A -85,B 0,C 180,E1 -22820.846,E2 -22820.846} C_VEL
LIN {X 0,Y 171.975,Z 440.644,A -85,B 0,C 180,E1 -22825.1,E2 -22825.1} C_VEL
LIN {X 0,Y 171.718,Z 438.741,A -85,B 0,C 180,E1 -22830.584,E2 -22830.584} C_VEL
LIN {X 0,Y 171.52,Z 437.21,A -85,B 0,C 180,E1 -22835.81,E2 -22835.81} C_VEL
LIN {X 0,Y 171.456,Z 436.63,A -85,B 0,C 180,E1 -22838.35,E2 -22838.35} C_VEL
LIN {X 0,Y 171.576,Z 436.614,A -85,B 0,C 180,E1 -22840.87,E2 -22840.87} C_VEL
LIN {X 0,Y 171.572,Z 436.614,A -85,B 0,C 180,E1 -22845.771,E2 -22845.771} C_VEL
LIN {X 0,Y 171.845,Z 436.579,A -85,B 0,C 180,E1 -22850.583,E2 -22850.583} C_VEL
LIN {X 0,Y 171.812,Z 436.582,A -85,B 0,C 180,E1 -22855.306,E2 -22855.306} C_VEL
LIN {X 0,Y 172.329,Z 436.492,A -85,B 0,C 180,E1 -22859.999,E2 -22859.999} C_VEL
LIN {X 0,Y 171.812,Z 436.57,A -85,B 0,C 180,E1 -22864.691,E2 -22864.691} C_VEL
LIN {X 0,Y 171.846,Z 436.571,A -85,B 0,C 180,E1 -22869.414,E2 -22869.414} C_VEL
LIN {X 0,Y 171.571,Z 436.606,A -85,B 0,C 180,E1 -22874.226,E2 -22874.226} C_VEL
LIN {X 0,Y 171.54,Z 436.608,A -85,B 0,C 180,E1 -22879.56,E2 -22879.56} C_VEL
LIN {X 0,Y 171.458,Z 436.621,A -85,B 0,C 180,E1 -22885.611,E2 -22885.611} C_VEL
LIN {X 0,Y 171.437,Z 436.63,A -85,B 0,C 180,E1 -22890.586,E2 -22890.586} C_VEL
LIN {X 0,Y 171.403,Z 436.634,A -85,B 0,C 180,E1 -22895.031,E2 -22895.031} C_VEL
LIN {X 0,Y 171.43,Z 436.631,A -85,B 0,C 180,E1 -22898.839,E2 -22898.839} C_VEL
LIN {X 0,Y 171.39,Z 436.731,A -85,B 0,C 180,E1 -22903.826,E2 -22903.826} C_VEL
LIN {X 0,Y 172.405,Z 439.503,A -85,B 0,C 180,E1 -22904.399,E2 -22904.399} C_VEL
LIN {X 0,Y 174.453,Z 441.984,A -85,B 0,C 180,E1 -22905.311,E2 -22905.311} C_VEL
LIN {X 0,Y 176.411,Z 445.331,A -85,B 0,C 180,E1 -22906.327,E2 -22906.327} C_VEL
LIN {X 0,Y 181.14,Z 453.49,A -85,B 0,C 180,E1 -22908.733,E2 -22908.733} C_VEL
LIN {X 0,Y 185.371,Z 462.288,A -85,B 0,C 180,E1 -22911.173,E2 -22911.173} C_VEL
LIN {X 0,Y 189.234,Z 472.182,A -85,B 0,C 180,E1 -22913.877,E2 -22913.877} C_VEL
LIN {X 0,Y 191.858,Z 480.79,A -85,B 0,C 180,E1 -22916.251,E2 -22916.251} C_VEL
LIN {X 0,Y 194.254,Z 490.781,A -85,B 0,C 180,E1 -22919.185,E2 -22919.185} C_VEL
LIN {X 0,Y 196.664,Z 498.06,A -85,B 0,C 180,E1 -22921.668,E2 -22921.668} C_VEL
LIN {X 0,Y 200.135,Z 505.3,A -85,B 0,C 180,E1 -22924.53,E2 -22924.53} C_VEL
LIN {X 0,Y 205.029,Z 512.297,A -85,B 0,C 180,E1 -22927.741,E2 -22927.741} C_VEL
LIN {X 0,Y 209.945,Z 517.489,A -85,B 0,C 180,E1 -22930.443,E2 -22930.443} C_VEL
LIN {X 0,Y 216.416,Z 522.726,A -85,B 0,C 180,E1 -22933.532,E2 -22933.532} C_VEL
LIN {X 0,Y 223.945,Z 527.254,A -85,B 0,C 180,E1 -22936.617,E2 -22936.617} C_VEL
LIN {X 0,Y 231.568,Z 530.903,A -85,B 0,C 180,E1 -22939.508,E2 -22939.508} C_VEL
LIN {X 0,Y 237,Z 533.019,A -85,B 0,C 180,E1 -22941.474,E2 -22941.474} C_VEL
LIN {X 0,Y 242.063,Z 534.674,A -85,B 0,C 180,E1 -22943.331,E2 -22943.331} C_VEL
LIN {X 0,Y 246.817,Z 536.024,A -85,B 0,C 180,E1 -22945.268,E2 -22945.268} C_VEL
LIN {X 0,Y 249.835,Z 536.831,A -85,B 0,C 180,E1 -22946.775,E2 -22946.775} C_VEL
LIN {X 0,Y 253.06,Z 537.414,A -85,B 0,C 180,E1 -22948.786,E2 -22948.786} C_VEL
LIN {X 0,Y 254.38,Z 537.468,A -85,B 0,C 180,E1 -22950,E2 -22950} C_VEL
LIN {X 0,Y 252.466,Z 537.337,A -85,B 0,C 180,E1 -22951.595,E2 -22951.595} C_VEL
LIN {X 0,Y 249.824,Z 536.83,A -85,B 0,C 180,E1 -22953.225,E2 -22953.225} C_VEL
LIN {X 0,Y 246.367,Z 535.916,A -85,B 0,C 180,E1 -22954.909,E2 -22954.909} C_VEL
LIN {X 0,Y 240.811,Z 534.277,A -85,B 0,C 180,E1 -22957.133,E2 -22957.133} C_VEL
LIN {X 0,Y 234.986,Z 532.252,A -85,B 0,C 180,E1 -22959.267,E2 -22959.267} C_VEL
LIN {X 0,Y 225.972,Z 528.339,A -85,B 0,C 180,E1 -22962.574,E2 -22962.574} C_VEL
LIN {X 0,Y 218.763,Z 524.257,A -85,B 0,C 180,E1 -22965.472,E2 -22965.472} C_VEL
LIN {X 0,Y 211.525,Z 518.899,A -85,B 0,C 180,E1 -22968.758,E2 -22968.758} C_VEL
LIN {X 0,Y 206.043,Z 513.529,A -85,B 0,C 180,E1 -22971.652,E2 -22971.652} C_VEL
LIN {X 0,Y 201.145,Z 506.845,A -85,B 0,C 180,E1 -22974.789,E2 -22974.789} C_VEL
LIN {X 0,Y 197.56,Z 500.15,A -85,B 0,C 180,E1 -22977.545,E2 -22977.545} C_VEL
LIN {X 0,Y 194.671,Z 492.193,A -85,B 0,C 180,E1 -22980.359,E2 -22980.359} C_VEL
LIN {X 0,Y 192.57,Z 483.676,A -85,B 0,C 180,E1 -22982.925,E2 -22982.925} C_VEL
LIN {X 0,Y 190.529,Z 476.102,A -85,B 0,C 180,E1 -22985.042,E2 -22985.042} C_VEL
LIN {X 0,Y 187.339,Z 467.001,A -85,B 0,C 180,E1 -22987.527,E2 -22987.527} C_VEL
LIN {X 0,Y 183.421,Z 458.136,A -85,B 0,C 180,E1 -22989.977,E2 -22989.977} C_VEL
LIN {X 0,Y 178.628,Z 449.114,A -85,B 0,C 180,E1 -22992.57,E2 -22992.57} C_VEL
LIN {X 0,Y 175.885,Z 444.734,A -85,B 0,C 180,E1 -22993.907,E2 -22993.907} C_VEL
LIN {X 0,Y 173.992,Z 441.31,A -85,B 0,C 180,E1 -22994.913,E2 -22994.913} C_VEL
LIN {X 0,Y 172.079,Z 439.018,A -85,B 0,C 180,E1 -22995.77,E2 -22995.77} C_VEL
LIN {X 0,Y 171.312,Z 436.646,A -85,B 0,C 180,E1 -22996.286,E2 -22996.286} C_VEL
LIN {X 0,Y 171.353,Z 436.64,A -85,B 0,C 180,E1 -23001.193,E2 -23001.193} C_VEL
LIN {X 0,Y 171.394,Z 436.636,A -85,B 0,C 180,E1 -23005.093,E2 -23005.093} C_VEL
LIN {X 0,Y 171.445,Z 436.63,A -85,B 0,C 180,E1 -23010.535,E2 -23010.535} C_VEL
LIN {X 0,Y 171.448,Z 436.622,A -85,B 0,C 180,E1 -23015.802,E2 -23015.802} C_VEL
LIN {X 0,Y 171.575,Z 436.605,A -85,B 0,C 180,E1 -23020.873,E2 -23020.873} C_VEL
LIN {X 0,Y 171.571,Z 436.606,A -85,B 0,C 180,E1 -23025.774,E2 -23025.774} C_VEL
LIN {X 0,Y 171.844,Z 436.571,A -85,B 0,C 180,E1 -23030.586,E2 -23030.586} C_VEL
LIN {X 0,Y 171.81,Z 436.57,A -85,B 0,C 180,E1 -23035.309,E2 -23035.309} C_VEL
LIN {X 0,Y 172.329,Z 436.492,A -85,B 0,C 180,E1 -23040.001,E2 -23040.001} C_VEL
LIN {X 0,Y 171.812,Z 436.583,A -85,B 0,C 180,E1 -23044.694,E2 -23044.694} C_VEL
LIN {X 0,Y 171.845,Z 436.58,A -85,B 0,C 180,E1 -23049.417,E2 -23049.417} C_VEL
LIN {X 0,Y 171.572,Z 436.617,A -85,B 0,C 180,E1 -23054.229,E2 -23054.229} C_VEL
LIN {X 0,Y 171.54,Z 436.618,A -85,B 0,C 180,E1 -23059.56,E2 -23059.56} C_VEL
LIN {X 0,Y 171.456,Z 436.629,A -85,B 0,C 180,E1 -23061.65,E2 -23061.65} C_VEL
LIN {X 0,Y 171.616,Z 437.931,A -85,B 0,C 180,E1 -23066.775,E2 -23066.775} C_VEL
LIN {X 0,Y 171.81,Z 439.653,A -85,B 0,C 180,E1 -23072.127,E2 -23072.127} C_VEL
LIN {X 0,Y 171.979,Z 440.749,A -85,B 0,C 180,E1 -23075.185,E2 -23075.185} C_VEL
LIN {X 0,Y 172.195,Z 442.262,A -85,B 0,C 180,E1 -23079.154,E2 -23079.154} C_VEL
LIN {X 0,Y 172.315,Z 444.419,A -85,B 0,C 180,E1 -23084.208,E2 -23084.208} C_VEL
LIN {X 0,Y 173.33,Z 447.509,A -85,B 0,C 180,E1 -23084.811,E2 -23084.811} C_VEL
LIN {X 0,Y 174.791,Z 450.075,A -85,B 0,C 180,E1 -23085.558,E2 -23085.558} C_VEL
LIN {X 0,Y 178.431,Z 459.078,A -85,B 0,C 180,E1 -23087.692,E2 -23087.692} C_VEL
LIN {X 0,Y 181.676,Z 470.277,A -85,B 0,C 180,E1 -23090.249,E2 -23090.249} C_VEL
LIN {X 0,Y 183.556,Z 480.621,A -85,B 0,C 180,E1 -23092.608,E2 -23092.608} C_VEL
LIN {X 0,Y 184.483,Z 489.756,A -85,B 0,C 180,E1 -23094.8,E2 -23094.8} C_VEL
LIN {X 0,Y 184.723,Z 498.79,A -85,B 0,C 180,E1 -23097.147,E2 -23097.147} C_VEL
LIN {X 0,Y 184.426,Z 505.545,A -85,B 0,C 180,E1 -23099.04,E2 -23099.04} C_VEL
LIN {X 0,Y 183.86,Z 509.41,A -85,B 0,C 180,E1 -23100.204,E2 -23100.204} C_VEL
LIN {X 0,Y 180.658,Z 517.961,A -85,B 0,C 180,E1 -23102.8,E2 -23102.8} C_VEL
LIN {X 0,Y 177.38,Z 526.387,A -85,B 0,C 180,E1 -23106.09,E2 -23106.09} C_VEL
LIN {X 0,Y 174.95,Z 531.949,A -85,B 0,C 180,E1 -23108.805,E2 -23108.805} C_VEL
LIN {X 0,Y 172.6,Z 537.442,A -85,B 0,C 180,E1 -23112.219,E2 -23112.219} C_VEL
LIN {X 0,Y 170.84,Z 541.771,A -85,B 0,C 180,E1 -23115.71,E2 -23115.71} C_VEL
LIN {X 0,Y 170.059,Z 544.143,A -85,B 0,C 180,E1 -23118.075,E2 -23118.075} C_VEL
LIN {X 0,Y 169.077,Z 547.34,A -85,B 0,C 180,E1 -23122.837,E2 -23122.837} C_VEL
LIN {X 0,Y 168.933,Z 548.406,A -85,B 0,C 180,E1 -23125.227,E2 -23125.227} C_VEL
LIN {X 0,Y 168.87,Z 548.999,A -85,B 0,C 180,E1 -23127.615,E2 -23127.615} C_VEL
LIN {X 0,Y 168.972,Z 549.158,A -85,B 0,C 180,E1 -23130,E2 -23130} C_VEL
LIN {X 0,Y 168.853,Z 548.939,A -85,B 0,C 180,E1 -23132.627,E2 -23132.627} C_VEL
LIN {X 0,Y 168.868,Z 548.404,A -85,B 0,C 180,E1 -23134.775,E2 -23134.775} C_VEL
LIN {X 0,Y 169.436,Z 545.947,A -85,B 0,C 180,E1 -23139.55,E2 -23139.55} C_VEL
LIN {X 0,Y 170.436,Z 542.991,A -85,B 0,C 180,E1 -23143.108,E2 -23143.108} C_VEL
LIN {X 0,Y 171.893,Z 538.996,A -85,B 0,C 180,E1 -23146.63,E2 -23146.63} C_VEL
LIN {X 0,Y 174.158,Z 533.867,A -85,B 0,C 180,E1 -23150.06,E2 -23150.06} C_VEL
LIN {X 0,Y 176.441,Z 528.606,A -85,B 0,C 180,E1 -23152.852,E2 -23152.852} C_VEL
LIN {X 0,Y 178.891,Z 522.285,A -85,B 0,C 180,E1 -23155.604,E2 -23155.604} C_VEL
LIN {X 0,Y 181.22,Z 516.333,A -85,B 0,C 180,E1 -23157.734,E2 -23157.734} C_VEL
LIN {X 0,Y 183.829,Z 509.409,A -85,B 0,C 180,E1 -23159.801,E2 -23159.801} C_VEL
LIN {X 0,Y 184.611,Z 502.31,A -85,B 0,C 180,E1 -23161.884,E2 -23161.884} C_VEL
LIN {X 0,Y 184.66,Z 493.579,A -85,B 0,C 180,E1 -23164.235,E2 -23164.235} C_VEL
LIN {X 0,Y 184.568,Z 491.298,A -85,B 0,C 180,E1 -23164.807,E2 -23164.807} C_VEL
LIN {X 0,Y 183.773,Z 486.954,A -85,B 0,C 180,E1 -23166.025,E2 -23166.025} C_VEL
LIN {X 0,Y 180.428,Z 480.561,A -85,B 0,C 180,E1 -23168.169,E2 -23168.169} C_VEL
LIN {X 0,Y 177.382,Z 475.508,A -85,B 0,C 180,E1 -23169.927,E2 -23169.927} C_VEL
LIN {X 0,Y 175.576,Z 471.315,A -85,B 0,C 180,E1 -23171.196,E2 -23171.196} C_VEL
LIN {X 0,Y 175.156,Z 469.786,A -85,B 0,C 180,E1 -23171.596,E2 -23171.596} C_VEL
LIN {X 0,Y 172.448,Z 460.72,A -85,B 0,C 180,E1 -23173.853,E2 -23173.853} C_VEL
LIN {X 0,Y 169.436,Z 453.274,A -85,B 0,C 180,E1 -23175.831,E2 -23175.831} C_VEL
LIN {X 0,Y 167.594,Z 449.185,A -85,B 0,C 180,E1 -23176.984,E2 -23176.984} C_VEL
LIN {X 0,Y 165.757,Z 446.304,A -85,B 0,C 180,E1 -23177.969,E2 -23177.969} C_VEL
LIN {X 0,Y 165.191,Z 444.082,A -85,B 0,C 180,E1 -23178.428,E2 -23178.428} C_VEL
LIN {X 0,Y 164.984,Z 442.227,A -85,B 0,C 180,E1 -23183.388,E2 -23183.388} C_VEL
LIN {X 0,Y 164.761,Z 440.267,A -85,B 0,C 180,E1 -23189.21,E2 -23189.21} C_VEL
LIN {X 0,Y 164.557,Z 438.614,A -85,B 0,C 180,E1 -23194.716,E2 -23194.716} C_VEL
LIN {X 0,Y 164.483,Z 437.499,A -85,B 0,C 180,E1 -23200.05,E2 -23200.05} C_VEL
LIN {X 0,Y 164.502,Z 437.494,A -85,B 0,C 180,E1 -23205.146,E2 -23205.146} C_VEL
LIN {X 0,Y 164.765,Z 437.461,A -85,B 0,C 180,E1 -23210.175,E2 -23210.175} C_VEL
LIN {X 0,Y 164.828,Z 437.451,A -85,B 0,C 180,E1 -23212.65,E2 -23212.65} C_VEL
LIN {X 0,Y 165.044,Z 437.424,A -85,B 0,C 180,E1 -23217.558,E2 -23217.558} C_VEL
LIN {X 0,Y 165.291,Z 437.367,A -85,B 0,C 180,E1 -23219.999,E2 -23219.999} C_VEL
LIN {X 0,Y 164.761,Z 437.45,A -85,B 0,C 180,E1 -23224.893,E2 -23224.893} C_VEL
LIN {X 0,Y 164.83,Z 437.453,A -85,B 0,C 180,E1 -23227.348,E2 -23227.348} C_VEL
LIN {X 0,Y 164.699,Z 437.466,A -85,B 0,C 180,E1 -23231.06,E2 -23231.06} C_VEL
LIN {X 0,Y 164.48,Z 437.497,A -85,B 0,C 180,E1 -23237.402,E2 -23237.402} C_VEL
LIN {X 0,Y 164.47,Z 437.488,A -85,B 0,C 180,E1 -23239.988,E2 -23239.988} C_VEL
LIN {X 0,Y 164.384,Z 437.504,A -85,B 0,C 180,E1 -23246.129,E2 -23246.129} C_VEL
LIN {X 0,Y 164.372,Z 437.509,A -85,B 0,C 180,E1 -23251.227,E2 -23251.227} C_VEL
LIN {X 0,Y 164.346,Z 437.514,A -85,B 0,C 180,E1 -23256.774,E2 -23256.774} C_VEL
LIN {X 0,Y 164.369,Z 437.511,A -85,B 0,C 180,E1 -23261.252,E2 -23261.252} C_VEL
LIN {X 0,Y 165.263,Z 440.193,A -85,B 0,C 180,E1 -23261.844,E2 -23261.844} C_VEL
LIN {X 0,Y 167.426,Z 442.745,A -85,B 0,C 180,E1 -23262.942,E2 -23262.942} C_VEL
LIN {X 0,Y 169.367,Z 446.158,A -85,B 0,C 180,E1 -23264.075,E2 -23264.075} C_VEL
LIN {X 0,Y 170.625,Z 448.129,A -85,B 0,C 180,E1 -23264.754,E2 -23264.754} C_VEL
LIN {X 0,Y 174.858,Z 455.533,A -85,B 0,C 180,E1 -23267.18,E2 -23267.18} C_VEL
LIN {X 0,Y 178.753,Z 463.424,A -85,B 0,C 180,E1 -23269.613,E2 -23269.613} C_VEL
LIN {X 0,Y 182.268,Z 472.234,A -85,B 0,C 180,E1 -23272.224,E2 -23272.224} C_VEL
LIN {X 0,Y 185.123,Z 481.303,A -85,B 0,C 180,E1 -23274.92,E2 -23274.92} C_VEL
LIN {X 0,Y 187.083,Z 490.016,A -85,B 0,C 180,E1 -23277.584,E2 -23277.584} C_VEL
LIN {X 0,Y 189.247,Z 498.172,A -85,B 0,C 180,E1 -23280.413,E2 -23280.413} C_VEL
LIN {X 0,Y 192.01,Z 505.016,A -85,B 0,C 180,E1 -23283.175,E2 -23283.175} C_VEL
LIN {X 0,Y 195.908,Z 511.677,A -85,B 0,C 180,E1 -23286.276,E2 -23286.276} C_VEL
LIN {X 0,Y 201.028,Z 517.746,A -85,B 0,C 180,E1 -23289.537,E2 -23289.537} C_VEL
LIN {X 0,Y 208.682,Z 524.045,A -85,B 0,C 180,E1 -23293.493,E2 -23293.493} C_VEL
LIN {X 0,Y 216.499,Z 528.605,A -85,B 0,C 180,E1 -23296.866,E2 -23296.866} C_VEL
LIN {X 0,Y 224.855,Z 532.275,A -85,B 0,C 180,E1 -23300.102,E2 -23300.102} C_VEL
LIN {X 0,Y 233.526,Z 535.082,A -85,B 0,C 180,E1 -23303.275,E2 -23303.275} C_VEL
LIN {X 0,Y 239.636,Z 536.584,A -85,B 0,C 180,E1 -23305.654,E2 -23305.654} C_VEL
LIN {X 0,Y 241.783,Z 537.056,A -85,B 0,C 180,E1 -23306.667,E2 -23306.667} C_VEL
LIN {X 0,Y 246.007,Z 537.645,A -85,B 0,C 180,E1 -23309.075,E2 -23309.075} C_VEL
LIN {X 0,Y 247.064,Z 537.667,A -85,B 0,C 180,E1 -23310,E2 -23310} C_VEL
LIN {X 0,Y 246.007,Z 537.646,A -85,B 0,C 180,E1 -23310.916,E2 -23310.916} C_VEL
LIN {X 0,Y 241.773,Z 537.056,A -85,B 0,C 180,E1 -23313.333,E2 -23313.333} C_VEL
LIN {X 0,Y 237.77,Z 536.152,A -85,B 0,C 180,E1 -23315.087,E2 -23315.087} C_VEL
LIN {X 0,Y 232.959,Z 534.93,A -85,B 0,C 180,E1 -23316.931,E2 -23316.931} C_VEL
LIN {X 0,Y 224.846,Z 532.275,A -85,B 0,C 180,E1 -23319.898,E2 -23319.898} C_VEL
LIN {X 0,Y 216.449,Z 528.607,A -85,B 0,C 180,E1 -23323.137,E2 -23323.137} C_VEL
LIN {X 0,Y 208.711,Z 524.049,A -85,B 0,C 180,E1 -23326.502,E2 -23326.502} C_VEL
LIN {X 0,Y 201.897,Z 518.565,A -85,B 0,C 180,E1 -23329.974,E2 -23329.974} C_VEL
LIN {X 0,Y 196.785,Z 512.813,A -85,B 0,C 180,E1 -23333.132,E2 -23333.132} C_VEL
LIN {X 0,Y 192.262,Z 505.559,A -85,B 0,C 180,E1 -23336.584,E2 -23336.584} C_VEL
LIN {X 0,Y 189.645,Z 499.26,A -85,B 0,C 180,E1 -23339.164,E2 -23339.164} C_VEL
LIN {X 0,Y 187.669,Z 492.412,A -85,B 0,C 180,E1 -23341.619,E2 -23341.619} C_VEL
LIN {X 0,Y 185.673,Z 483.486,A -85,B 0,C 180,E1 -23344.416,E2 -23344.416} C_VEL
LIN {X 0,Y 183.32,Z 475.366,A -85,B 0,C 180,E1 -23346.845,E2 -23346.845} C_VEL
LIN {X 0,Y 180.262,Z 466.967,A -85,B 0,C 180,E1 -23349.325,E2 -23349.325} C_VEL
LIN {X 0,Y 176.632,Z 459.026,A -85,B 0,C 180,E1 -23351.753,E2 -23351.753} C_VEL
LIN {X 0,Y 171.695,Z 450.01,A -85,B 0,C 180,E1 -23354.658,E2 -23354.658} C_VEL
LIN {X 0,Y 169.467,Z 446.331,A -85,B 0,C 180,E1 -23355.868,E2 -23355.868} C_VEL
LIN {X 0,Y 167.555,Z 443.242,A -85,B 0,C 180,E1 -23356.947,E2 -23356.947} C_VEL
LIN {X 0,Y 166.73,Z 442.017,A -85,B 0,C 180,E1 -23357.411,E2 -23357.411} C_VEL
LIN {X 0,Y 164.91,Z 439.696,A -85,B 0,C 180,E1 -23358.353,E2 -23358.353} C_VEL
LIN {X 0,Y 164.294,Z 437.52,A -85,B 0,C 180,E1 -23358.877,E2 -23358.877} C_VEL
LIN {X 0,Y 164.325,Z 437.514,A -85,B 0,C 180,E1 -23364.35,E2 -23364.35} C_VEL
LIN {X 0,Y 164.386,Z 437.507,A -85,B 0,C 180,E1 -23369.135,E2 -23369.135} C_VEL
LIN {X 0,Y 164.406,Z 437.497,A -85,B 0,C 180,E1 -23374.694,E2 -23374.694} C_VEL
LIN {X 0,Y 164.481,Z 437.487,A -85,B 0,C 180,E1 -23380.052,E2 -23380.052} C_VEL
LIN {X 0,Y 164.501,Z 437.485,A -85,B 0,C 180,E1 -23385.149,E2 -23385.149} C_VEL
LIN {X 0,Y 164.764,Z 437.453,A -85,B 0,C 180,E1 -23390.178,E2 -23390.178} C_VEL
LIN {X 0,Y 164.827,Z 437.454,A -85,B 0,C 180,E1 -23392.652,E2 -23392.652} C_VEL
LIN {X 0,Y 165.043,Z 437.389,A -85,B 0,C 180,E1 -23397.561,E2 -23397.561} C_VEL
LIN {X 0,Y 165.291,Z 437.367,A -85,B 0,C 180,E1 -23400.001,E2 -23400.001} C_VEL
LIN {X 0,Y 164.761,Z 437.462,A -85,B 0,C 180,E1 -23404.895,E2 -23404.895} C_VEL
LIN {X 0,Y 164.828,Z 437.454,A -85,B 0,C 180,E1 -23407.35,E2 -23407.35} C_VEL
LIN {X 0,Y 164.701,Z 437.47,A -85,B 0,C 180,E1 -23411.062,E2 -23411.062} C_VEL
LIN {X 0,Y 164.48,Z 437.499,A -85,B 0,C 180,E1 -23417.405,E2 -23417.405} C_VEL
LIN {X 0,Y 164.472,Z 437.498,A -85,B 0,C 180,E1 -23419.991,E2 -23419.991} C_VEL
LIN {X 0,Y 164.557,Z 438.61,A -85,B 0,C 180,E1 -23425.284,E2 -23425.284} C_VEL
LIN {X 0,Y 164.761,Z 440.265,A -85,B 0,C 180,E1 -23430.79,E2 -23430.79} C_VEL
LIN {X 0,Y 164.984,Z 442.227,A -85,B 0,C 180,E1 -23436.612,E2 -23436.612} C_VEL
LIN {X 0,Y 165.197,Z 444.052,A -85,B 0,C 180,E1 -23441.327,E2 -23441.327} C_VEL
LIN {X 0,Y 165.202,Z 444.182,A -85,B 0,C 180,E1 -23441.618,E2 -23441.618} C_VEL
LIN {X 0,Y 166.205,Z 447.233,A -85,B 0,C 180,E1 -23442.283,E2 -23442.283} C_VEL
LIN {X 0,Y 168.014,Z 449.98,A -85,B 0,C 180,E1 -23443.266,E2 -23443.266} C_VEL
LIN {X 0,Y 169.778,Z 453.842,A -85,B 0,C 180,E1 -23444.354,E2 -23444.354} C_VEL
LIN {X 0,Y 172.942,Z 461.952,A -85,B 0,C 180,E1 -23446.492,E2 -23446.492} C_VEL
LIN {X 0,Y 175.197,Z 469.88,A -85,B 0,C 180,E1 -23448.433,E2 -23448.433} C_VEL
LIN {X 0,Y 176.967,Z 478.551,A -85,B 0,C 180,E1 -23450.55,E2 -23450.55} C_VEL
LIN {X 0,Y 178.124,Z 489.503,A -85,B 0,C 180,E1 -23453.334,E2 -23453.334} C_VEL
LIN {X 0,Y 178.334,Z 497.575,A -85,B 0,C 180,E1 -23455.513,E2 -23455.513} C_VEL
LIN {X 0,Y 178.036,Z 505.337,A -85,B 0,C 180,E1 -23457.798,E2 -23457.798} C_VEL
LIN {X 0,Y 177.539,Z 509.206,A -85,B 0,C 180,E1 -23459.029,E2 -23459.029} C_VEL
LIN {X 0,Y 175.689,Z 514.511,A -85,B 0,C 180,E1 -23460.658,E2 -23460.658} C_VEL
LIN {X 0,Y 173.087,Z 520.711,A -85,B 0,C 180,E1 -23462.82,E2 -23462.82} C_VEL
LIN {X 0,Y 170.398,Z 527.252,A -85,B 0,C 180,E1 -23465.642,E2 -23465.642} C_VEL
LIN {X 0,Y 168.32,Z 531.751,A -85,B 0,C 180,E1 -23467.928,E2 -23467.928} C_VEL
LIN {X 0,Y 165.84,Z 537.245,A -85,B 0,C 180,E1 -23471.468,E2 -23471.468} C_VEL
LIN {X 0,Y 163.917,Z 541.572,A -85,B 0,C 180,E1 -23475.093,E2 -23475.093} C_VEL
LIN {X 0,Y 163.102,Z 543.946,A -85,B 0,C 180,E1 -23477.558,E2 -23477.558} C_VEL
LIN {X 0,Y 162.417,Z 545.749,A -85,B 0,C 180,E1 -23480.033,E2 -23480.033} C_VEL
LIN {X 0,Y 161.852,Z 548.208,A -85,B 0,C 180,E1 -23485.018,E2 -23485.018} C_VEL
LIN {X 0,Y 161.8,Z 548.803,A -85,B 0,C 180,E1 -23487.511,E2 -23487.511} C_VEL
LIN {X 0,Y 161.884,Z 548.961,A -85,B 0,C 180,E1 -23490,E2 -23490} C_VEL
LIN {X 0,Y 161.763,Z 548.802,A -85,B 0,C 180,E1 -23492.49,E2 -23492.49} C_VEL
LIN {X 0,Y 161.795,Z 548.207,A -85,B 0,C 180,E1 -23494.984,E2 -23494.984} C_VEL
LIN {X 0,Y 162.417,Z 545.749,A -85,B 0,C 180,E1 -23499.967,E2 -23499.967} C_VEL
LIN {X 0,Y 163.479,Z 542.793,A -85,B 0,C 180,E1 -23503.677,E2 -23503.677} C_VEL
LIN {X 0,Y 165.084,Z 538.798,A -85,B 0,C 180,E1 -23507.337,E2 -23507.337} C_VEL
LIN {X 0,Y 167.464,Z 533.669,A -85,B 0,C 180,E1 -23510.898,E2 -23510.898} C_VEL
LIN {X 0,Y 169.902,Z 528.409,A -85,B 0,C 180,E1 -23513.785,E2 -23513.785} C_VEL
LIN {X 0,Y 172.484,Z 522.087,A -85,B 0,C 180,E1 -23516.628,E2 -23516.628} C_VEL
LIN {X 0,Y 174.944,Z 516.135,A -85,B 0,C 180,E1 -23518.82,E2 -23518.82} C_VEL
LIN {X 0,Y 177.006,Z 511.131,A -85,B 0,C 180,E1 -23520.413,E2 -23520.413} C_VEL
LIN {X 0,Y 177.744,Z 507.271,A -85,B 0,C 180,E1 -23521.594,E2 -23521.594} C_VEL
LIN {X 0,Y 178.282,Z 500.955,A -85,B 0,C 180,E1 -23523.496,E2 -23523.496} C_VEL
LIN {X 0,Y 178.282,Z 492.348,A -85,B 0,C 180,E1 -23525.9,E2 -23525.9} C_VEL
LIN {X 0,Y 177.585,Z 483.57,A -85,B 0,C 180,E1 -23528.185,E2 -23528.185} C_VEL
LIN {X 0,Y 176.312,Z 474.876,A -85,B 0,C 180,E1 -23530.327,E2 -23530.327} C_VEL
LIN {X 0,Y 175.156,Z 469.786,A -85,B 0,C 180,E1 -23531.596,E2 -23531.596} C_VEL
LIN {X 0,Y 173.934,Z 467.079,A -85,B 0,C 180,E1 -23532.442,E2 -23532.442} C_VEL
LIN {X 0,Y 170.593,Z 463.822,A -85,B 0,C 180,E1 -23534.021,E2 -23534.021} C_VEL
LIN {X 0,Y 166.285,Z 460.098,A -85,B 0,C 180,E1 -23536.021,E2 -23536.021} C_VEL
LIN {X 0,Y 165.193,Z 458.446,A -85,B 0,C 180,E1 -23536.659,E2 -23536.659} C_VEL
LIN {X 0,Y 162.933,Z 453.724,A -85,B 0,C 180,E1 -23538.144,E2 -23538.144} C_VEL
LIN {X 0,Y 161.213,Z 450.235,A -85,B 0,C 180,E1 -23539.294,E2 -23539.294} C_VEL
LIN {X 0,Y 160.527,Z 448.96,A -85,B 0,C 180,E1 -23539.75,E2 -23539.75} C_VEL
LIN {X 0,Y 158.554,Z 445.887,A -85,B 0,C 180,E1 -23540.953,E2 -23540.953} C_VEL
LIN {X 0,Y 157.994,Z 443.792,A -85,B 0,C 180,E1 -23541.481,E2 -23541.481} C_VEL
LIN {X 0,Y 157.86,Z 442.725,A -85,B 0,C 180,E1 -23544.634,E2 -23544.634} C_VEL
LIN {X 0,Y 157.739,Z 441.703,A -85,B 0,C 180,E1 -23547.835,E2 -23547.835} C_VEL
LIN {X 0,Y 157.606,Z 440.038,A -85,B 0,C 180,E1 -23553.516,E2 -23553.516} C_VEL
LIN {X 0,Y 157.422,Z 438.511,A -85,B 0,C 180,E1 -23559.638,E2 -23559.638} C_VEL
LIN {X 0,Y 157.439,Z 438.374,A -85,B 0,C 180,E1 -23564.463,E2 -23564.463} C_VEL
LIN {X 0,Y 157.687,Z 438.344,A -85,B 0,C 180,E1 -23569.729,E2 -23569.729} C_VEL
LIN {X 0,Y 157.765,Z 438.331,A -85,B 0,C 180,E1 -23572.318,E2 -23572.318} C_VEL
LIN {X 0,Y 158.254,Z 438.242,A -85,B 0,C 180,E1 -23579.999,E2 -23579.999} C_VEL
LIN {X 0,Y 157.766,Z 438.332,A -85,B 0,C 180,E1 -23587.679,E2 -23587.679} C_VEL
LIN {X 0,Y 157.634,Z 438.347,A -85,B 0,C 180,E1 -23591.236,E2 -23591.236} C_VEL
LIN {X 0,Y 157.438,Z 438.366,A -85,B 0,C 180,E1 -23595.534,E2 -23595.534} C_VEL
LIN {X 0,Y 157.366,Z 438.376,A -85,B 0,C 180,E1 -23600.932,E2 -23600.932} C_VEL
LIN {X 0,Y 157.307,Z 438.389,A -85,B 0,C 180,E1 -23606.681,E2 -23606.681} C_VEL
LIN {X 0,Y 157.274,Z 438.395,A -85,B 0,C 180,E1 -23612.426,E2 -23612.426} C_VEL
LIN {X 0,Y 157.29,Z 438.392,A -85,B 0,C 180,E1 -23617.474,E2 -23617.474} C_VEL
LIN {X 0,Y 157.274,Z 438.392,A -85,B 0,C 180,E1 -23618.255,E2 -23618.255} C_VEL
LIN {X 0,Y 158.211,Z 441.121,A -85,B 0,C 180,E1 -23618.967,E2 -23618.967} C_VEL
LIN {X 0,Y 160.663,Z 443.944,A -85,B 0,C 180,E1 -23620.411,E2 -23620.411} C_VEL
LIN {X 0,Y 162.458,Z 447.104,A -85,B 0,C 180,E1 -23621.587,E2 -23621.587} C_VEL
LIN {X 0,Y 163.614,Z 448.705,A -85,B 0,C 180,E1 -23622.259,E2 -23622.259} C_VEL
LIN {X 0,Y 165.853,Z 452.194,A -85,B 0,C 180,E1 -23623.593,E2 -23623.593} C_VEL
LIN {X 0,Y 171.594,Z 463.422,A -85,B 0,C 180,E1 -23627.494,E2 -23627.494} C_VEL
LIN {X 0,Y 175.329,Z 472.314,A -85,B 0,C 180,E1 -23630.407,E2 -23630.407} C_VEL
LIN {X 0,Y 178.189,Z 481.322,A -85,B 0,C 180,E1 -23633.283,E2 -23633.283} C_VEL
LIN {X 0,Y 180.031,Z 488.807,A -85,B 0,C 180,E1 -23635.713,E2 -23635.713} C_VEL
LIN {X 0,Y 182.058,Z 498.69,A -85,B 0,C 180,E1 -23639.22,E2 -23639.22} C_VEL
LIN {X 0,Y 184.586,Z 505.855,A -85,B 0,C 180,E1 -23642.241,E2 -23642.241} C_VEL
LIN {X 0,Y 187.636,Z 511.809,A -85,B 0,C 180,E1 -23645.112,E2 -23645.112} C_VEL
LIN {X 0,Y 192.385,Z 517.997,A -85,B 0,C 180,E1 -23648.574,E2 -23648.574} C_VEL
LIN {X 0,Y 196.84,Z 522.264,A -85,B 0,C 180,E1 -23651.257,E2 -23651.257} C_VEL
LIN {X 0,Y 203.861,Z 527.201,A -85,B 0,C 180,E1 -23654.854,E2 -23654.854} C_VEL
LIN {X 0,Y 212.523,Z 531.431,A -85,B 0,C 180,E1 -23658.556,E2 -23658.556} C_VEL
LIN {X 0,Y 220.271,Z 534.196,A -85,B 0,C 180,E1 -23661.52,E2 -23661.52} C_VEL
LIN {X 0,Y 228.896,Z 536.396,A -85,B 0,C 180,E1 -23664.715,E2 -23664.715} C_VEL
LIN {X 0,Y 233.589,Z 537.285,A -85,B 0,C 180,E1 -23666.55,E2 -23666.55} C_VEL
LIN {X 0,Y 237,Z 537.764,A -85,B 0,C 180,E1 -23668.301,E2 -23668.301} C_VEL
LIN {X 0,Y 239.728,Z 537.867,A -85,B 0,C 180,E1 -23670,E2 -23670} C_VEL
LIN {X 0,Y 236.993,Z 537.764,A -85,B 0,C 180,E1 -23671.699,E2 -23671.699} C_VEL
LIN {X 0,Y 232.457,Z 537.103,A -85,B 0,C 180,E1 -23673.898,E2 -23673.898} C_VEL
LIN {X 0,Y 226.246,Z 535.85,A -85,B 0,C 180,E1 -23676.274,E2 -23676.274} C_VEL
LIN {X 0,Y 218.126,Z 533.55,A -85,B 0,C 180,E1 -23679.27,E2 -23679.27} C_VEL
LIN {X 0,Y 209.056,Z 529.943,A -85,B 0,C 180,E1 -23682.865,E2 -23682.865} C_VEL
LIN {X 0,Y 201.741,Z 525.871,A -85,B 0,C 180,E1 -23686.182,E2 -23686.182} C_VEL
LIN {X 0,Y 194.52,Z 520.235,A -85,B 0,C 180,E1 -23690.056,E2 -23690.056} C_VEL
LIN {X 0,Y 189.116,Z 513.892,A -85,B 0,C 180,E1 -23693.76,E2 -23693.76} C_VEL
LIN {X 0,Y 185.26,Z 507.322,A -85,B 0,C 180,E1 -23697.079,E2 -23697.079} C_VEL
LIN {X 0,Y 182.732,Z 500.605,A -85,B 0,C 180,E1 -23699.999,E2 -23699.999} C_VEL
LIN {X 0,Y 181.183,Z 494.626,A -85,B 0,C 180,E1 -23702.298,E2 -23702.298} C_VEL
LIN {X 0,Y 179.189,Z 484.926,A -85,B 0,C 180,E1 -23705.53,E2 -23705.53} C_VEL
LIN {X 0,Y 176.739,Z 476.522,A -85,B 0,C 180,E1 -23708.25,E2 -23708.25} C_VEL
LIN {X 0,Y 173.943,Z 468.759,A -85,B 0,C 180,E1 -23710.751,E2 -23710.751} C_VEL
LIN {X 0,Y 170.017,Z 460.141,A -85,B 0,C 180,E1 -23713.637,E2 -23713.637} C_VEL
LIN {X 0,Y 165.808,Z 452.299,A -85,B 0,C 180,E1 -23716.406,E2 -23716.406} C_VEL
LIN {X 0,Y 163.378,Z 448.4,A -85,B 0,C 180,E1 -23717.874,E2 -23717.874} C_VEL
LIN {X 0,Y 160.784,Z 444.548,A -85,B 0,C 180,E1 -23719.453,E2 -23719.453} C_VEL
LIN {X 0,Y 160.145,Z 443.273,A -85,B 0,C 180,E1 -23719.905,E2 -23719.905} C_VEL
LIN {X 0,Y 158.068,Z 441.003,A -85,B 0,C 180,E1 -23721.112,E2 -23721.112} C_VEL
LIN {X 0,Y 157.207,Z 438.401,A -85,B 0,C 180,E1 -23721.89,E2 -23721.89} C_VEL
LIN {X 0,Y 157.274,Z 438.392,A -85,B 0,C 180,E1 -23724.486,E2 -23724.486} C_VEL
LIN {X 0,Y 157.289,Z 438.393,A -85,B 0,C 180,E1 -23728.097,E2 -23728.097} C_VEL
LIN {X 0,Y 157.313,Z 438.387,A -85,B 0,C 180,E1 -23733.466,E2 -23733.466} C_VEL
LIN {X 0,Y 157.39,Z 438.371,A -85,B 0,C 180,E1 -23739.669,E2 -23739.669} C_VEL
LIN {X 0,Y 157.438,Z 438.366,A -85,B 0,C 180,E1 -23744.466,E2 -23744.466} C_VEL
LIN {X 0,Y 157.685,Z 438.335,A -85,B 0,C 180,E1 -23749.732,E2 -23749.732} C_VEL
LIN {X 0,Y 157.764,Z 438.332,A -85,B 0,C 180,E1 -23752.321,E2 -23752.321} C_VEL
LIN {X 0,Y 158.254,Z 438.242,A -85,B 0,C 180,E1 -23760.001,E2 -23760.001} C_VEL
LIN {X 0,Y 157.765,Z 438.334,A -85,B 0,C 180,E1 -23767.682,E2 -23767.682} C_VEL
LIN {X 0,Y 157.635,Z 438.351,A -85,B 0,C 180,E1 -23771.238,E2 -23771.238} C_VEL
LIN {X 0,Y 157.439,Z 438.377,A -85,B 0,C 180,E1 -23775.537,E2 -23775.537} C_VEL
LIN {X 0,Y 157.422,Z 438.509,A -85,B 0,C 180,E1 -23780.362,E2 -23780.362} C_VEL
LIN {X 0,Y 157.606,Z 440.036,A -85,B 0,C 180,E1 -23786.484,E2 -23786.484} C_VEL
LIN {X 0,Y 157.741,Z 441.752,A -85,B 0,C 180,E1 -23792.322,E2 -23792.322} C_VEL
LIN {X 0,Y 157.947,Z 443.204,A -85,B 0,C 180,E1 -23796.783,E2 -23796.783} C_VEL
LIN {X 0,Y 158.045,Z 444.082,A -85,B 0,C 180,E1 -23798.643,E2 -23798.643} C_VEL
LIN {X 0,Y 159.078,Z 446.93,A -85,B 0,C 180,E1 -23799.377,E2 -23799.377} C_VEL
LIN {X 0,Y 161.162,Z 450.01,A -85,B 0,C 180,E1 -23800.655,E2 -23800.655} C_VEL
LIN {X 0,Y 162.813,Z 453.577,A -85,B 0,C 180,E1 -23801.79,E2 -23801.79} C_VEL
LIN {X 0,Y 163.813,Z 455.375,A -85,B 0,C 180,E1 -23802.407,E2 -23802.407} C_VEL
LIN {X 0,Y 166.826,Z 462.942,A -85,B 0,C 180,E1 -23804.667,E2 -23804.667} C_VEL
LIN {X 0,Y 169.131,Z 470.727,A -85,B 0,C 180,E1 -23806.8,E2 -23806.8} C_VEL
LIN {X 0,Y 170.876,Z 479.17,A -85,B 0,C 180,E1 -23809.047,E2 -23809.047} C_VEL
LIN {X 0,Y 171.829,Z 489.283,A -85,B 0,C 180,E1 -23811.755,E2 -23811.755} C_VEL
LIN {X 0,Y 172.047,Z 497.304,A -85,B 0,C 180,E1 -23814.043,E2 -23814.043} C_VEL
LIN {X 0,Y 171.715,Z 505.13,A -85,B 0,C 180,E1 -23816.461,E2 -23816.461} C_VEL
LIN {X 0,Y 170.854,Z 510.932,A -85,B 0,C 180,E1 -23818.368,E2 -23818.368} C_VEL
LIN {X 0,Y 166.773,Z 520.513,A -85,B 0,C 180,E1 -23821.701,E2 -23821.701} C_VEL
LIN {X 0,Y 163.923,Z 527.054,A -85,B 0,C 180,E1 -23824.613,E2 -23824.613} C_VEL
LIN {X 0,Y 161.745,Z 531.554,A -85,B 0,C 180,E1 -23826.98,E2 -23826.98} C_VEL
LIN {X 0,Y 159.086,Z 537.047,A -85,B 0,C 180,E1 -23830.651,E2 -23830.651} C_VEL
LIN {X 0,Y 157.02,Z 541.374,A -85,B 0,C 180,E1 -23834.422,E2 -23834.422} C_VEL
LIN {X 0,Y 156.126,Z 543.747,A -85,B 0,C 180,E1 -23836.993,E2 -23836.993} C_VEL
LIN {X 0,Y 155.42,Z 545.552,A -85,B 0,C 180,E1 -23839.579,E2 -23839.579} C_VEL
LIN {X 0,Y 154.754,Z 548.011,A -85,B 0,C 180,E1 -23844.789,E2 -23844.789} C_VEL
LIN {X 0,Y 154.715,Z 548.727,A -85,B 0,C 180,E1 -23847.983,E2 -23847.983} C_VEL
LIN {X 0,Y 154.687,Z 548.756,A -85,B 0,C 180,E1 -23851.695,E2 -23851.695} C_VEL
LIN {X 0,Y 154.715,Z 548.01,A -85,B 0,C 180,E1 -23855.212,E2 -23855.212} C_VEL
LIN {X 0,Y 155.42,Z 545.552,A -85,B 0,C 180,E1 -23860.421,E2 -23860.421} C_VEL
LIN {X 0,Y 156.549,Z 542.594,A -85,B 0,C 180,E1 -23864.295,E2 -23864.295} C_VEL
LIN {X 0,Y 158.308,Z 538.601,A -85,B 0,C 180,E1 -23868.105,E2 -23868.105} C_VEL
LIN {X 0,Y 160.801,Z 533.47,A -85,B 0,C 180,E1 -23871.808,E2 -23871.808} C_VEL
LIN {X 0,Y 163.405,Z 528.211,A -85,B 0,C 180,E1 -23874.793,E2 -23874.793} C_VEL
LIN {X 0,Y 165.614,Z 523.087,A -85,B 0,C 180,E1 -23877.229,E2 -23877.229} C_VEL
LIN {X 0,Y 168.054,Z 517.564,A -85,B 0,C 180,E1 -23879.431,E2 -23879.431} C_VEL
LIN {X 0,Y 170.828,Z 510.931,A -85,B 0,C 180,E1 -23881.637,E2 -23881.637} C_VEL
LIN {X 0,Y 171.851,Z 503.035,A -85,B 0,C 180,E1 -23884.215,E2 -23884.215} C_VEL
LIN {X 0,Y 172.026,Z 493.502,A -85,B 0,C 180,E1 -23887.055,E2 -23887.055} C_VEL
LIN {X 0,Y 171.388,Z 483.723,A -85,B 0,C 180,E1 -23889.746,E2 -23889.746} C_VEL
LIN {X 0,Y 170.136,Z 475.426,A -85,B 0,C 180,E1 -23891.964,E2 -23891.964} C_VEL
LIN {X 0,Y 167.746,Z 465.65,A -85,B 0,C 180,E1 -23894.581,E2 -23894.581} C_VEL
LIN {X 0,Y 165.193,Z 458.446,A -85,B 0,C 180,E1 -23896.659,E2 -23896.659} C_VEL
LIN {X 0,Y 163.341,Z 456.321,A -85,B 0,C 180,E1 -23897.67,E2 -23897.67} C_VEL
LIN {X 0,Y 155.617,Z 452.253,A -85,B 0,C 180,E1 -23901.426,E2 -23901.426} C_VEL
LIN {X 0,Y 154.376,Z 450.297,A -85,B 0,C 180,E1 -23902.284,E2 -23902.284} C_VEL
LIN {X 0,Y 154.218,Z 449.804,A -85,B 0,C 180,E1 -23902.434,E2 -23902.434} C_VEL
LIN {X 0,Y 151.577,Z 446.11,A -85,B 0,C 180,E1 -23904.272,E2 -23904.272} C_VEL
LIN {X 0,Y 150.788,Z 443.532,A -85,B 0,C 180,E1 -23904.978,E2 -23904.978} C_VEL
LIN {X 0,Y 150.642,Z 442.305,A -85,B 0,C 180,E1 -23909.122,E2 -23909.122} C_VEL
LIN {X 0,Y 150.569,Z 441.375,A -85,B 0,C 180,E1 -23912.478,E2 -23912.478} C_VEL
LIN {X 0,Y 150.388,Z 440.007,A -85,B 0,C 180,E1 -23918.045,E2 -23918.045} C_VEL
LIN {X 0,Y 150.369,Z 439.378,A -85,B 0,C 180,E1 -23920.902,E2 -23920.902} C_VEL
LIN {X 0,Y 150.428,Z 439.248,A -85,B 0,C 180,E1 -23926.489,E2 -23926.489} C_VEL
LIN {X 0,Y 150.609,Z 439.225,A -85,B 0,C 180,E1 -23929.241,E2 -23929.241} C_VEL
LIN {X 0,Y 150.702,Z 439.212,A -85,B 0,C 180,E1 -23931.956,E2 -23931.956} C_VEL
LIN {X 0,Y 151.214,Z 439.117,A -85,B 0,C 180,E1 -23939.999,E2 -23939.999} C_VEL
LIN {X 0,Y 150.703,Z 439.21,A -85,B 0,C 180,E1 -23948.041,E2 -23948.041} C_VEL
LIN {X 0,Y 150.574,Z 439.227,A -85,B 0,C 180,E1 -23951.436,E2 -23951.436} C_VEL
LIN {X 0,Y 150.35,Z 439.254,A -85,B 0,C 180,E1 -23956.286,E2 -23956.286} C_VEL
LIN {X 0,Y 150.347,Z 439.249,A -85,B 0,C 180,E1 -23960.791,E2 -23960.791} C_VEL
LIN {X 0,Y 150.238,Z 439.272,A -85,B 0,C 180,E1 -23967.279,E2 -23967.279} C_VEL
LIN {X 0,Y 150.214,Z 439.274,A -85,B 0,C 180,E1 -23972.634,E2 -23972.634} C_VEL
LIN {X 0,Y 150.214,Z 439.275,A -85,B 0,C 180,E1 -23974.763,E2 -23974.763} C_VEL
LIN {X 0,Y 151.097,Z 441.84,A -85,B 0,C 180,E1 -23975.548,E2 -23975.548} C_VEL
LIN {X 0,Y 153.189,Z 444.178,A -85,B 0,C 180,E1 -23976.991,E2 -23976.991} C_VEL
LIN {X 0,Y 153.88,Z 445.237,A -85,B 0,C 180,E1 -23977.501,E2 -23977.501} C_VEL
LIN {X 0,Y 155.633,Z 448.124,A -85,B 0,C 180,E1 -23978.779,E2 -23978.779} C_VEL
LIN {X 0,Y 156.866,Z 449.667,A -85,B 0,C 180,E1 -23979.569,E2 -23979.569} C_VEL
LIN {X 0,Y 161.783,Z 458.056,A -85,B 0,C 180,E1 -23983.085,E2 -23983.085} C_VEL
LIN {X 0,Y 166.48,Z 467.781,A -85,B 0,C 180,E1 -23986.735,E2 -23986.735} C_VEL
LIN {X 0,Y 169.542,Z 475.59,A -85,B 0,C 180,E1 -23989.518,E2 -23989.518} C_VEL
LIN {X 0,Y 171.889,Z 483.225,A -85,B 0,C 180,E1 -23992.172,E2 -23992.172} C_VEL
LIN {X 0,Y 173.517,Z 490.155,A -85,B 0,C 180,E1 -23994.596,E2 -23994.596} C_VEL
LIN {X 0,Y 175.175,Z 499.478,A -85,B 0,C 180,E1 -23998.075,E2 -23998.075} C_VEL
LIN {X 0,Y 177.015,Z 505.884,A -85,B 0,C 180,E1 -24000.861,E2 -24000.861} C_VEL
LIN {X 0,Y 179.804,Z 512.207,A -85,B 0,C 180,E1 -24004.024,E2 -24004.024} C_VEL
LIN {X 0,Y 183.854,Z 518.247,A -85,B 0,C 180,E1 -24007.527,E2 -24007.527} C_VEL
LIN {X 0,Y 189.332,Z 523.711,A -85,B 0,C 180,E1 -24011.219,E2 -24011.219} C_VEL
LIN {X 0,Y 196.408,Z 528.52,A -85,B 0,C 180,E1 -24015.041,E2 -24015.041} C_VEL
LIN {X 0,Y 202.959,Z 531.697,A -85,B 0,C 180,E1 -24018.009,E2 -24018.009} C_VEL
LIN {X 0,Y 208.603,Z 533.818,A -85,B 0,C 180,E1 -24020.302,E2 -24020.302} C_VEL
LIN {X 0,Y 214.247,Z 535.452,A -85,B 0,C 180,E1 -24022.46,E2 -24022.46} C_VEL
LIN {X 0,Y 219.735,Z 536.648,A -85,B 0,C 180,E1 -24024.494,E2 -24024.494} C_VEL
LIN {X 0,Y 225.294,Z 537.578,A -85,B 0,C 180,E1 -24026.575,E2 -24026.575} C_VEL
LIN {X 0,Y 228.983,Z 537.985,A -85,B 0,C 180,E1 -24028.241,E2 -24028.241} C_VEL
LIN {X 0,Y 232.247,Z 538.071,A -85,B 0,C 180,E1 -24030,E2 -24030} C_VEL
LIN {X 0,Y 228.959,Z 537.986,A -85,B 0,C 180,E1 -24031.759,E2 -24031.759} C_VEL
LIN {X 0,Y 224.84,Z 537.529,A -85,B 0,C 180,E1 -24033.584,E2 -24033.584} C_VEL
LIN {X 0,Y 218.981,Z 536.502,A -85,B 0,C 180,E1 -24035.79,E2 -24035.79} C_VEL
LIN {X 0,Y 212.922,Z 535.084,A -85,B 0,C 180,E1 -24038.028,E2 -24038.028} C_VEL
LIN {X 0,Y 207.122,Z 533.336,A -85,B 0,C 180,E1 -24040.264,E2 -24040.264} C_VEL
LIN {X 0,Y 197.534,Z 529.138,A -85,B 0,C 180,E1 -24044.421,E2 -24044.421} C_VEL
LIN {X 0,Y 191.581,Z 525.445,A -85,B 0,C 180,E1 -24047.491,E2 -24047.491} C_VEL
LIN {X 0,Y 185.808,Z 520.423,A -85,B 0,C 180,E1 -24051.073,E2 -24051.073} C_VEL
LIN {X 0,Y 181.285,Z 514.622,A -85,B 0,C 180,E1 -24054.629,E2 -24054.629} C_VEL
LIN {X 0,Y 178.286,Z 509.132,A -85,B 0,C 180,E1 -24057.591,E2 -24057.591} C_VEL
LIN {X 0,Y 175.541,Z 500.83,A -85,B 0,C 180,E1 -24061.363,E2 -24061.363} C_VEL
LIN {X 0,Y 174.023,Z 492.848,A -85,B 0,C 180,E1 -24064.429,E2 -24064.429} C_VEL
LIN {X 0,Y 172.556,Z 485.797,A -85,B 0,C 180,E1 -24066.94,E2 -24066.94} C_VEL
LIN {X 0,Y 169.998,Z 476.919,A -85,B 0,C 180,E1 -24070.026,E2 -24070.026} C_VEL
LIN {X 0,Y 167.248,Z 469.478,A -85,B 0,C 180,E1 -24072.661,E2 -24072.661} C_VEL
LIN {X 0,Y 162.648,Z 459.87,A -85,B 0,C 180,E1 -24076.264,E2 -24076.264} C_VEL
LIN {X 0,Y 157.764,Z 451.496,A -85,B 0,C 180,E1 -24079.766,E2 -24079.766} C_VEL
LIN {X 0,Y 156.087,Z 448.707,A -85,B 0,C 180,E1 -24080.925,E2 -24080.925} C_VEL
LIN {X 0,Y 154,Z 445.757,A -85,B 0,C 180,E1 -24082.359,E2 -24082.359} C_VEL
LIN {X 0,Y 153.295,Z 444.31,A -85,B 0,C 180,E1 -24082.935,E2 -24082.935} C_VEL
LIN {X 0,Y 151.091,Z 441.876,A -85,B 0,C 180,E1 -24084.45,E2 -24084.45} C_VEL
LIN {X 0,Y 150.207,Z 439.276,A -85,B 0,C 180,E1 -24085.337,E2 -24085.337} C_VEL
LIN {X 0,Y 150.203,Z 439.274,A -85,B 0,C 180,E1 -24089.025,E2 -24089.025} C_VEL
LIN {X 0,Y 150.238,Z 439.272,A -85,B 0,C 180,E1 -24092.721,E2 -24092.721} C_VEL
LIN {X 0,Y 150.347,Z 439.249,A -85,B 0,C 180,E1 -24099.209,E2 -24099.209} C_VEL
LIN {X 0,Y 150.35,Z 439.254,A -85,B 0,C 180,E1 -24103.714,E2 -24103.714} C_VEL
LIN {X 0,Y 150.607,Z 439.219,A -85,B 0,C 180,E1 -24109.244,E2 -24109.244} C_VEL
LIN {X 0,Y 150.701,Z 439.21,A -85,B 0,C 180,E1 -24111.959,E2 -24111.959} C_VEL
LIN {X 0,Y 151.214,Z 439.117,A -85,B 0,C 180,E1 -24120.001,E2 -24120.001} C_VEL
LIN {X 0,Y 150.702,Z 439.215,A -85,B 0,C 180,E1 -24128.044,E2 -24128.044} C_VEL
LIN {X 0,Y 150.575,Z 439.231,A -85,B 0,C 180,E1 -24131.438,E2 -24131.438} C_VEL
LIN {X 0,Y 150.35,Z 439.259,A -85,B 0,C 180,E1 -24136.289,E2 -24136.289} C_VEL
LIN {X 0,Y 150.369,Z 439.377,A -85,B 0,C 180,E1 -24139.098,E2 -24139.098} C_VEL
LIN {X 0,Y 150.469,Z 440.695,A -85,B 0,C 180,E1 -24144.859,E2 -24144.859} C_VEL
LIN {X 0,Y 150.568,Z 441.458,A -85,B 0,C 180,E1 -24147.826,E2 -24147.826} C_VEL
LIN {X 0,Y 150.718,Z 442.914,A -85,B 0,C 180,E1 -24152.932,E2 -24152.932} C_VEL
LIN {X 0,Y 150.807,Z 443.649,A -85,B 0,C 180,E1 -24155.017,E2 -24155.017} C_VEL
LIN {X 0,Y 151.983,Z 446.866,A -85,B 0,C 180,E1 -24156.027,E2 -24156.027} C_VEL
LIN {X 0,Y 154.277,Z 449.975,A -85,B 0,C 180,E1 -24157.621,E2 -24157.621} C_VEL
LIN {X 0,Y 156.159,Z 453.825,A -85,B 0,C 180,E1 -24159.057,E2 -24159.057} C_VEL
LIN {X 0,Y 157.11,Z 455.441,A -85,B 0,C 180,E1 -24159.707,E2 -24159.707} C_VEL
LIN {X 0,Y 160.039,Z 462.075,A -85,B 0,C 180,E1 -24162.045,E2 -24162.045} C_VEL
LIN {X 0,Y 162.598,Z 469.557,A -85,B 0,C 180,E1 -24164.399,E2 -24164.399} C_VEL
LIN {X 0,Y 164.458,Z 478.089,A -85,B 0,C 180,E1 -24166.864,E2 -24166.864} C_VEL
LIN {X 0,Y 165.517,Z 486.443,A -85,B 0,C 180,E1 -24169.267,E2 -24169.267} C_VEL
LIN {X 0,Y 165.829,Z 497.084,A -85,B 0,C 180,E1 -24172.468,E2 -24172.468} C_VEL
LIN {X 0,Y 165.385,Z 505.452,A -85,B 0,C 180,E1 -24175.198,E2 -24175.198} C_VEL
LIN {X 0,Y 164.645,Z 510.728,A -85,B 0,C 180,E1 -24177.028,E2 -24177.028} C_VEL
LIN {X 0,Y 162.679,Z 515.742,A -85,B 0,C 180,E1 -24178.775,E2 -24178.775} C_VEL
LIN {X 0,Y 159.857,Z 521.691,A -85,B 0,C 180,E1 -24181.08,E2 -24181.08} C_VEL
LIN {X 0,Y 157.502,Z 526.856,A -85,B 0,C 180,E1 -24183.499,E2 -24183.499} C_VEL
LIN {X 0,Y 155.226,Z 531.357,A -85,B 0,C 180,E1 -24185.954,E2 -24185.954} C_VEL
LIN {X 0,Y 152.377,Z 536.849,A -85,B 0,C 180,E1 -24189.763,E2 -24189.763} C_VEL
LIN {X 0,Y 150.152,Z 541.176,A -85,B 0,C 180,E1 -24193.69,E2 -24193.69} C_VEL
LIN {X 0,Y 149.173,Z 543.549,A -85,B 0,C 180,E1 -24196.375,E2 -24196.375} C_VEL
LIN {X 0,Y 148.407,Z 545.354,A -85,B 0,C 180,E1 -24199.081,E2 -24199.081} C_VEL
LIN {X 0,Y 147.687,Z 547.814,A -85,B 0,C 180,E1 -24204.539,E2 -24204.539} C_VEL
LIN {X 0,Y 147.628,Z 548.565,A -85,B 0,C 180,E1 -24208.728,E2 -24208.728} C_VEL
LIN {X 0,Y 147.572,Z 548.407,A -85,B 0,C 180,E1 -24212.73,E2 -24212.73} C_VEL
LIN {X 0,Y 147.638,Z 547.812,A -85,B 0,C 180,E1 -24215.463,E2 -24215.463} C_VEL
LIN {X 0,Y 148.407,Z 545.354,A -85,B 0,C 180,E1 -24220.919,E2 -24220.919} C_VEL
LIN {X 0,Y 149.645,Z 542.396,A -85,B 0,C 180,E1 -24224.969,E2 -24224.969} C_VEL
LIN {X 0,Y 151.563,Z 538.403,A -85,B 0,C 180,E1 -24228.94,E2 -24228.94} C_VEL
LIN {X 0,Y 154.189,Z 533.272,A -85,B 0,C 180,E1 -24232.794,E2 -24232.794} C_VEL
LIN {X 0,Y 156.938,Z 528.012,A -85,B 0,C 180,E1 -24235.888,E2 -24235.888} C_VEL
LIN {X 0,Y 159.196,Z 523.096,A -85,B 0,C 180,E1 -24238.316,E2 -24238.316} C_VEL
LIN {X 0,Y 161.879,Z 517.366,A -85,B 0,C 180,E1 -24240.672,E2 -24240.672} C_VEL
LIN {X 0,Y 164.097,Z 512.487,A -85,B 0,C 180,E1 -24242.367,E2 -24242.367} C_VEL
LIN {X 0,Y 165.153,Z 507.123,A -85,B 0,C 180,E1 -24244.22,E2 -24244.22} C_VEL
LIN {X 0,Y 165.727,Z 499.38,A -85,B 0,C 180,E1 -24246.797,E2 -24246.797} C_VEL
LIN {X 0,Y 165.754,Z 492.047,A -85,B 0,C 180,E1 -24249.062,E2 -24249.062} C_VEL
LIN {X 0,Y 165.199,Z 483.442,A -85,B 0,C 180,E1 -24251.569,E2 -24251.569} C_VEL
LIN {X 0,Y 163.677,Z 474.225,A -85,B 0,C 180,E1 -24254.233,E2 -24254.233} C_VEL
LIN {X 0,Y 161.475,Z 465.936,A -85,B 0,C 180,E1 -24256.723,E2 -24256.723} C_VEL
LIN {X 0,Y 158.665,Z 458.718,A -85,B 0,C 180,E1 -24259.119,E2 -24259.119} C_VEL
LIN {X 0,Y 156.386,Z 454.097,A -85,B 0,C 180,E1 -24260.802,E2 -24260.802} C_VEL
LIN {X 0,Y 154.348,Z 450.239,A -85,B 0,C 180,E1 -24262.306,E2 -24262.306} C_VEL
LIN {X 0,Y 154.218,Z 449.804,A -85,B 0,C 180,E1 -24262.434,E2 -24262.434} C_VEL
LIN {X 0,Y 153.076,Z 447.215,A -85,B 0,C 180,E1 -24263.393,E2 -24263.393} C_VEL
LIN {X 0,Y 150.631,Z 444.669,A -85,B 0,C 180,E1 -24265.134,E2 -24265.134} C_VEL
LIN {X 0,Y 147.973,Z 443.363,A -85,B 0,C 180,E1 -24267.094,E2 -24267.094} C_VEL
LIN {X 0,Y 144.837,Z 442.85,A -85,B 0,C 180,E1 -24270.082,E2 -24270.082} C_VEL
LIN {X 0,Y 143.568,Z 442.406,A -85,B 0,C 180,E1 -24272.48,E2 -24272.48} C_VEL
LIN {X 0,Y 143.46,Z 442.211,A -85,B 0,C 180,E1 -24273.299,E2 -24273.299} C_VEL
LIN {X 0,Y 143.385,Z 440.981,A -85,B 0,C 180,E1 -24278.633,E2 -24278.633} C_VEL
LIN {X 0,Y 143.297,Z 440.141,A -85,B 0,C 180,E1 -24282.885,E2 -24282.885} C_VEL
LIN {X 0,Y 143.535,Z 440.107,A -85,B 0,C 180,E1 -24288.704,E2 -24288.704} C_VEL
LIN {X 0,Y 143.623,Z 440.095,A -85,B 0,C 180,E1 -24291.557,E2 -24291.557} C_VEL
LIN {X 0,Y 144.173,Z 439.992,A -85,B 0,C 180,E1 -24299.998,E2 -24299.998} C_VEL
LIN {X 0,Y 143.624,Z 440.088,A -85,B 0,C 180,E1 -24308.44,E2 -24308.44} C_VEL
LIN {X 0,Y 143.502,Z 440.109,A -85,B 0,C 180,E1 -24311.628,E2 -24311.628} C_VEL
LIN {X 0,Y 143.293,Z 440.136,A -85,B 0,C 180,E1 -24317.113,E2 -24317.113} C_VEL
LIN {X 0,Y 143.273,Z 440.133,A -85,B 0,C 180,E1 -24321.253,E2 -24321.253} C_VEL
LIN {X 0,Y 143.185,Z 440.149,A -85,B 0,C 180,E1 -24327.935,E2 -24327.935} C_VEL
LIN {X 0,Y 143.136,Z 440.154,A -85,B 0,C 180,E1 -24330.521,E2 -24330.521} C_VEL
LIN {X 0,Y 143.979,Z 442.677,A -85,B 0,C 180,E1 -24331.443,E2 -24331.443} C_VEL
LIN {X 0,Y 146.078,Z 445.058,A -85,B 0,C 180,E1 -24333.209,E2 -24333.209} C_VEL
LIN {X 0,Y 146.91,Z 445.858,A -85,B 0,C 180,E1 -24333.852,E2 -24333.852} C_VEL
LIN {X 0,Y 148.757,Z 449.099,A -85,B 0,C 180,E1 -24335.464,E2 -24335.464} C_VEL
LIN {X 0,Y 150.198,Z 450.816,A -85,B 0,C 180,E1 -24336.52,E2 -24336.52} C_VEL
LIN {X 0,Y 151.811,Z 453.625,A -85,B 0,C 180,E1 -24337.873,E2 -24337.873} C_VEL
LIN {X 0,Y 152.664,Z 454.631,A -85,B 0,C 180,E1 -24338.502,E2 -24338.502} C_VEL
LIN {X 0,Y 157.791,Z 464.259,A -85,B 0,C 180,E1 -24342.782,E2 -24342.782} C_VEL
LIN {X 0,Y 161.112,Z 471.557,A -85,B 0,C 180,E1 -24345.739,E2 -24345.739} C_VEL
LIN {X 0,Y 164.463,Z 480.922,A -85,B 0,C 180,E1 -24349.359,E2 -24349.359} C_VEL
LIN {X 0,Y 166.734,Z 490.039,A -85,B 0,C 180,E1 -24352.803,E2 -24352.803} C_VEL
LIN {X 0,Y 168.135,Z 498.533,A -85,B 0,C 180,E1 -24356.12,E2 -24356.12} C_VEL
LIN {X 0,Y 169.311,Z 504.629,A -85,B 0,C 180,E1 -24358.746,E2 -24358.746} C_VEL
LIN {X 0,Y 171.915,Z 512.209,A -85,B 0,C 180,E1 -24362.62,E2 -24362.62} C_VEL
LIN {X 0,Y 175.526,Z 518.493,A -85,B 0,C 180,E1 -24366.398,E2 -24366.398} C_VEL
LIN {X 0,Y 179.792,Z 523.292,A -85,B 0,C 180,E1 -24369.739,E2 -24369.739} C_VEL
LIN {X 0,Y 186.157,Z 528.174,A -85,B 0,C 180,E1 -24373.723,E2 -24373.723} C_VEL
LIN {X 0,Y 194.168,Z 532.276,A -85,B 0,C 180,E1 -24377.756,E2 -24377.756} C_VEL
LIN {X 0,Y 199.726,Z 534.328,A -85,B 0,C 180,E1 -24380.146,E2 -24380.146} C_VEL
LIN {X 0,Y 205.591,Z 535.939,A -85,B 0,C 180,E1 -24382.448,E2 -24382.448} C_VEL
LIN {X 0,Y 211.727,Z 537.144,A -85,B 0,C 180,E1 -24384.742,E2 -24384.742} C_VEL
LIN {X 0,Y 218.137,Z 537.981,A -85,B 0,C 180,E1 -24387.129,E2 -24387.129} C_VEL
LIN {X 0,Y 220.654,Z 538.215,A -85,B 0,C 180,E1 -24388.175,E2 -24388.175} C_VEL
LIN {X 0,Y 224.403,Z 538.284,A -85,B 0,C 180,E1 -24390,E2 -24390} C_VEL
LIN {X 0,Y 220.625,Z 538.216,A -85,B 0,C 180,E1 -24391.825,E2 -24391.825} C_VEL
LIN {X 0,Y 215.8,Z 537.781,A -85,B 0,C 180,E1 -24393.734,E2 -24393.734} C_VEL
LIN {X 0,Y 210.366,Z 536.905,A -85,B 0,C 180,E1 -24395.752,E2 -24395.752} C_VEL
LIN {X 0,Y 204.672,Z 535.716,A -85,B 0,C 180,E1 -24397.894,E2 -24397.894} C_VEL
LIN {X 0,Y 198.926,Z 534.091,A -85,B 0,C 180,E1 -24400.174,E2 -24400.174} C_VEL
LIN {X 0,Y 188.969,Z 529.819,A -85,B 0,C 180,E1 -24404.771,E2 -24404.771} C_VEL
LIN {X 0,Y 183.458,Z 526.399,A -85,B 0,C 180,E1 -24407.846,E2 -24407.846} C_VEL
LIN {X 0,Y 177.338,Z 520.702,A -85,B 0,C 180,E1 -24412.114,E2 -24412.114} C_VEL
LIN {X 0,Y 173.227,Z 514.856,A -85,B 0,C 180,E1 -24415.86,E2 -24415.86} C_VEL
LIN {X 0,Y 170.592,Z 508.879,A -85,B 0,C 180,E1 -24419.157,E2 -24419.157} C_VEL
LIN {X 0,Y 168.563,Z 501.052,A -85,B 0,C 180,E1 -24422.82,E2 -24422.82} C_VEL
LIN {X 0,Y 167.351,Z 493.072,A -85,B 0,C 180,E1 -24426.01,E2 -24426.01} C_VEL
LIN {X 0,Y 166.019,Z 486.719,A -85,B 0,C 180,E1 -24428.454,E2 -24428.454} C_VEL
LIN {X 0,Y 163.629,Z 478.379,A -85,B 0,C 180,E1 -24431.611,E2 -24431.611} C_VEL
LIN {X 0,Y 160.731,Z 470.621,A -85,B 0,C 180,E1 -24434.636,E2 -24434.636} C_VEL
LIN {X 0,Y 156.327,Z 461.451,A -85,B 0,C 180,E1 -24438.481,E2 -24438.481} C_VEL
LIN {X 0,Y 152.56,Z 454.636,A -85,B 0,C 180,E1 -24441.547,E2 -24441.547} C_VEL
LIN {X 0,Y 150.354,Z 451.326,A -85,B 0,C 180,E1 -24443.316,E2 -24443.316} C_VEL
LIN {X 0,Y 149.485,Z 449.888,A -85,B 0,C 180,E1 -24444.009,E2 -24444.009} C_VEL
LIN {X 0,Y 147.363,Z 446.998,A -85,B 0,C 180,E1 -24445.682,E2 -24445.682} C_VEL
LIN {X 0,Y 146.551,Z 445.375,A -85,B 0,C 180,E1 -24446.448,E2 -24446.448} C_VEL
LIN {X 0,Y 144.236,Z 443.121,A -85,B 0,C 180,E1 -24448.312,E2 -24448.312} C_VEL
LIN {X 0,Y 143.202,Z 440.573,A -85,B 0,C 180,E1 -24449.393,E2 -24449.393} C_VEL
LIN {X 0,Y 143.132,Z 440.155,A -85,B 0,C 180,E1 -24449.58,E2 -24449.58} C_VEL
